Omron CX-Programmer project NewProject (CX-Programmer 9.61)

# PLC NewPLC1: CJ2M CPU31
I/O table (CPU CJ2M-CPU31): rack 0 slot 0 CJ1W-ID211; rack 0 slot 1 CJ1W-ID211; rack 0 slot 2 CJ1W-ID211; rack 0 slot 3 CJ1W-OD211; rack 0 slot 4 CJ1W-OD211; rack 0 slot 5 CJ1W-OD211; rack 0 slot 11 CJ2M-EIP21

## Global symbols (name address type ; comment)
0.00 BOOL  ; MASTER ON
0.01 BOOL  ; SW AUT/MAN
0.02 BOOL  ; PB START
0.03 BOOL  ; PB_EXECUTE
0.04 BOOL  ; PB RESET
0.06 BOOL  ; IN INV1 FAULT
0.07 BOOL  ; IN INV2 FAULT
0.08 BOOL  ; IN INV3 FAULT
0.09 BOOL  ; IN INV4 FAULT
0.10 BOOL  ; IN INV5 FAULT
0.11 BOOL  ; RUN INV1
0.12 BOOL  ; RUN INV2
0.13 BOOL  ; RUN INV3
0.14 BOOL  ; RUN INV4
0.15 BOOL  ; RUN INV5
10.00 BOOL  ; IR HMI PB FWD MOTOR 1
10.01 BOOL  ; IR HMI PB RVS MOTOR 1
10.02 BOOL  ; IR HMI PB FWD MOTOR2
10.03 BOOL  ; IR HMI PB RVS MOTOR2
10.04 BOOL  ; IR HMI PB STRAIGHT
10.05 BOOL  ; IR HMI PB TURN
10.06 BOOL  ; IR HMI PB FWD MOTOR4
10.07 BOOL  ; IR HMI PB RVS MOTOR4
10.08 BOOL  ; IR HMI PB FWD MOTOR5
10.09 BOOL  ; IR HMI PB RVS MOTOR 5
10.10 BOOL  ; IR HMI PB STP1 UP
10.11 BOOL  ; IR HMI PB STP1 DN
10.12 BOOL  ; IR HMI PB STP2 UP
10.13 BOOL  ; IR HMI PB STP2 DN
10.14 BOOL  ; IR HMI PB STP3 UP
10.15 BOOL  ; IR HMI PB STP3 DN
11.00 BOOL  ; AUTO READY
11.01 BOOL  ; MANUAL READY
11.04 BOOL  ; SET RFID ENABLED
11.05 BOOL  ; STRAIGHT CONV CONFIRM
11.06 BOOL  ; TURNING CONV CONFIRM
11.09 BOOL  ; 16.06
11.10 BOOL  ; DELETE ALL DATA
11.11 BOOL  ; ON/OFF YELLOW LAMP
11.13 BOOL  ; MATERIAL CANNOT ENTER SEGMEN 2
11.14 BOOL  ; DELETE 1 MEMORY ROTATE
11.15 BOOL  ; DELETE 1 MEMORY STRAIGHT
12.00 BOOL  ; MASTER OFF
13.02 BOOL  ; ROT_CONV_NEXT DATA
13.03 BOOL  ; ROT_CONV_PREV DATA
14.00 BOOL  ; IR MAN M1 FWD
14.01 BOOL  ; IR MAN M1 RVS
14.02 BOOL  ; IR MAN M2 FWD
14.03 BOOL  ; IR MAN M2 RVS
14.04 BOOL  ; IR MAN STRAIGHT ROT
14.05 BOOL  ; IR MAN TURN ROT
14.06 BOOL  ; IR MAN M4 FWD
14.07 BOOL  ; IR MAN M4 RVS
14.08 BOOL  ; IR MAN M5 FWD
14.09 BOOL  ; IR MAN M5 RVS
14.10 BOOL  ; IR MAN STP1 UP
14.11 BOOL  ; IR MAN STP1 DN
14.12 BOOL  ; IR MAN STP2 UP
14.13 BOOL  ; IR MAN STP2 DN
14.14 BOOL  ; IR MAN STP3 UP
14.15 BOOL  ; IR MAN STP3 DN
15.00 BOOL  ; IR RS UP STP1
15.01 BOOL  ; IR RS DN STP1
15.02 BOOL  ; IR RS UP STP2
15.03 BOOL  ; IR RS DN STP2
15.04 BOOL  ; IR RS UP STP3
15.05 BOOL  ; IR RS DN STP3
15.06 BOOL  ; IR FAULT CONFIRM
15.07 BOOL  ; IR OUT M1 FWD
15.08 BOOL  ; IR OUT M1 RVS
15.09 BOOL  ; IR OUT M2 FWD
15.10 BOOL  ; IR OUT M2 RVS
15.11 BOOL  ; IR OUT M3 FWD
15.12 BOOL  ; IR OUT M3 RVS
15.13 BOOL  ; IR OUT M4 FWD
15.14 BOOL  ; IR OUT M4 RVS
15.15 BOOL  ; IR OUT M5 FWD
16.00 BOOL  ; IR OUT M5 RVS
16.01 BOOL  ; IR PH1
16.02 BOOL  ; IR PH2
16.03 BOOL  ; IR PH3
16.04 BOOL  ; IR PH4
16.05 BOOL  ; IR PH5
16.06 BOOL  ; IR PH6
16.07 BOOL  ; IR PH7
16.08 BOOL  ; IR PH8
16.09 BOOL  ; IR PH9
16.10 BOOL  ; AUTO M1 FWD
16.11 BOOL  ; AUTO M2 FWD IN MATERIAL
16.12 BOOL  ; AUTO STP1 DOWN
16.13 BOOL  ; AUTO M2 FWD OUT MATERIAL
16.14 BOOL  ; AUTO STP1 UP
16.15 BOOL  ; AUTO STP2 DOWN
17.00 BOOL  ; AUTO ROLLER ROTARY FWD IN MATERIAL
17.01 BOOL  ; AUTO STP3 DOWN
17.02 BOOL  ; AUTO ROLLER ROTARY FWD OUT MATERIAL
17.03 BOOL  ; AUTO STP3 UP
17.04 BOOL  ; AUTO M4 FWD IN MATERIAL
17.06 BOOL  ; AUTO M5 FWD IN MATERIAL
17.07 BOOL  ; HOMEPOST
17.08 BOOL  ; IR MANUAL MODE
17.09 BOOL  ; AUTO STP2 UP
17.10 BOOL  ; MATERIAL STRAIGHT
17.11 BOOL  ; MATERIAL TURN
17.12 BOOL  ; IR RS UP STP ROTARY
17.13 BOOL  ; IR RS DN STP ROTARY
17.14 BOOL  ; IR LS TURN
17.15 BOOL  ; IR LS STRAIGHT
18.00 BOOL  ; IR HMI INDI M3 FWD
18.01 BOOL  ; IR HMI INDI M3 RVS
18.02 BOOL  ; IR HMI PB STP ROT UP
18.03 BOOL  ; IR HMI STP ROT DN
18.04 BOOL  ; IR MAN STP ROT UP
18.05 BOOL  ; IR MAN STP ROT DN
18.06 BOOL  ; AUTO DN STP ROTARY
18.07 BOOL  ; AUTO M3 TURN
18.08 BOOL  ; AUTO STP ROTARY UP
18.09 BOOL  ; CONFIRM BASE TURN
18.10 BOOL  ; AUTO STP2 DOWN TURN
18.11 BOOL  ; CONFIRM TRANFER MATERIAL
18.12 BOOL  ; AUTO STP ROT DN
18.13 BOOL  ; AUTO STP2 UP AFTER TRANSFER TURN
18.14 BOOL  ; AUTO M3 BACK STRAIGHT
18.15 BOOL  ; AUTO STP ROT UP AFTER TRANFER TURN
19.00 BOOL  ; MAN ROTARY TURN
19.01 BOOL  ; MAN ROTARY STRAIGHT
19.02 BOOL  ; STP ROT UP
19.03 BOOL  ; STP ROT UP
19.04 BOOL  ; IR MAN M ROLLER RVS
19.05 BOOL  ; IR MAN M ROLLER FWD
19.06 BOOL  ; IR HMI PB M ROLLER FWD
19.07 BOOL  ; IR HMI PB M ROLLER RVS
19.08 BOOL  ; SET LS STRAIGHT
19.09 BOOL  ; SET LS TURN
19.10 BOOL  ; SET STP ROT UP
19.11 BOOL  ; SET STP ROT UP
19.12 BOOL  ; SET STP ROT DN
19.13 BOOL  ; AUTO DELAY OFF M1
19.14 BOOL  ; SET HOMEPOST ALL
19.15 BOOL  ; AUTO ROLLER ROT RVS TRANFER MATERIAL
1.00 BOOL  ; PH1
1.01 BOOL  ; PH2
1.02 BOOL  ; PH3
1.03 BOOL  ; PH4
1.04 BOOL  ; EMERGENCY SHUTTER
1.05 BOOL  ; AIR PRESURE ON
1.06 BOOL  ; PH5
1.07 BOOL  ; RS UP STP2
1.08 BOOL  ; RS DN STP2
1.09 BOOL  ; PH6
1.10 BOOL  ; RS DN STP3
1.11 BOOL  ; RS UP STP3
1.12 BOOL  ; RS UP STP ROTARY
1.13 BOOL  ; RS DN STP ROTARY
1.14 BOOL  ; LS TURN
1.15 BOOL  ; LS STRAIGHT
20.00 BOOL  ; SAVE 1
20.01 BOOL  ; SAVE 2
20.02 BOOL  ; HMI IN NO BLOWING
20.03 BOOL  ; CONFIRM NO BLOWING
20.04 BOOL  ; AIR SOURCE OFF CONFIRM
20.05 BOOL  ; SET DELAY STP3 UP
20.06 BOOL  ; DON'T CONFIRM
20.07 BOOL  ; ROT RUN TURN
20.08 BOOL  ; SET OF M5
20.09 BOOL  ; SET OFF M1
20.10 BOOL  ; LONG MATERIAL WAITING IN ROTARY
20.11 BOOL  ; DELAY OFF RVS ROLLER
20.12 BOOL  ; IR LAST DATA
20.13 BOOL  ; MATERIAL WAIT ON CONV 1
20.14 BOOL  ; STP2 UP WAIT LONG MATERIAL
20.15 BOOL  ; STP2 CAN'T UP
2.00 BOOL  ; PH7
2.01 BOOL  ; PH8
2.02 BOOL  ; PH9
2.03 BOOL  ; PH9
2.04 BOOL  ; INTERLOCK BLOWING DOOR NOT OPEN
2.05 BOOL  ; INTERLOCK BLOWING PHOTOSENSOR
2.12 BOOL  ; RS DN STP1
2.13 BOOL  ; RS UP STP1
3.00 BOOL  ; SOL UP STP1
3.01 BOOL  ; SOL DN STP1
3.02 BOOL  ; SOL UP STP2
3.03 BOOL  ; SOL DN STP2
3.04 BOOL  ; SOL UP STP3
3.05 BOOL  ; SOL DN STP3
3.08 BOOL  ; TOWER LAMP GREEN
3.09 BOOL  ; TOWER LAMP YELLOW
3.10 BOOL  ; TOWER LAMP RED
3.11 BOOL  ; OUT RESET INV1
3.12 BOOL  ; OUT RESET INV2
3.13 BOOL  ; OUT RESET INV3
3.14 BOOL  ; OUT RESET INV4
3.15 BOOL  ; OUT RESET INV5
4.00 BOOL  ; BUZZER
4.01 BOOL  ; AUTORUN LAMP
4.02 BOOL  ; INDILAMP YELLOW
4.03 BOOL  ; FAULT LAMP
4.04 BOOL  ; OUT M1 FWD
4.05 BOOL  ; OUT M1 RVS
4.06 BOOL  ; OUT M2 FWD
4.07 BOOL  ; OUT M2 RVS
4.08 BOOL  ; OUT M3 TURN
4.09 BOOL  ; OUT M3 STRAIGHT
4.10 BOOL  ; OUT M4 FWD
4.11 BOOL  ; OUT M4 RVS
4.12 BOOL  ; OUT M5 FWD
4.13 BOOL  ; OUT M5 RVS
4.14 BOOL  ; KONTAKTOR M4
4.15 BOOL  ; KONTAKTOR M5
5.00 BOOL  ; SOL UP STP ROT
5.01 BOOL  ; SOL DN STP ROT
5.02 BOOL  ; OUT RELAY BRAKE
5.03 BOOL  ; OUT M ROLLER FWD
5.04 BOOL  ; OUT M ROLLER RVS
5.05 BOOL  ; BLOWING NO ROTATE
5.15 BOOL  ; chiyoda
99.00 BOOL  ; MASTER ON
99.01 BOOL  ; MASTER OFF
99.02 BOOL  ; IR_FAULT_CONFIRM
D1000 CHANNEL  ; READ DATA FROM RFID
D1002 CHANNEL  ; INPUT DATA WORD 1
D1003 CHANNEL  ; INPUT DATA WORD 2
D1010 CHANNEL  ; ID RECODED 1
D1011 CHANNEL  ; ID RECORDED2
D1093 CHANNEL  ; STACK LOCATION
D1450 CHANNEL  ; DATA INDIRECT
D1460 CHANNEL  ; DATA INDIRECT
D1800 CHANNEL  ; DATA INPUT
D1820 CHANNEL  ; DATA INPUT
D2000 CHANNEL  ; MEMORY 1 NO BLOWING
D2002 CHANNEL  ; MEEMORY 2 NO BLOWING
D2004 CHANNEL  ; MEMORY NO 3 NO BLOWING
D2006 CHANNEL  ; MEMORY 4 NO BLOWING
D2008 CHANNEL  ; MEMORY 5 NO BLOWING
D2010 CHANNEL  ; MEMORY 6 NO BLOWING
D2012 CHANNEL  ; MEMORY 7 NO BLOWING
D2014 CHANNEL  ; MEMORY 8 NO BLOWING
D2016 CHANNEL  ; MEMORY 9 NO BLOWING
D2018 CHANNEL  ; MEMORY 10 NO BLOWING
D3000 CHANNEL  ; LAST DATA ACTION
D50 CHANNEL  ; ID RECORDED1
D51 CHANNEL  ; ID RECORDED2
D90 CHANNEL  ; DATA STRAIGHT STACK
D91 CHANNEL  ; DATA 2X STRAIGHT STACK
T0001 BOOL  ; DELAY ON M1
T0002 BOOL  ; DELAY OFF M1
T0003 BOOL  ; DELAY OFF M2 OUT MATERIAL
T0004 BOOL  ; DELAY DOWN STP3
T0005 BOOL  ; DELAY OFF MOTOR ROLLER
T0006 BOOL  ; DELAY UP STP 3
T0007 BOOL  ; DELAY STP1 DOWN
T0008 BOOL  ; DELAY TURN
T0009 BOOL  ; DELAY STP3 UP
T0010 BOOL  ; DELAY SAFETY OFF BY SELF
T0011 BOOL  ; DELAY SAFETY OFF BY SELF M2
T0012 BOOL  ; DELAY SAFETY OFF BY SELF
T0013 BOOL  ; DELAY OFF BUTTON NO ROTATE BLOWING
T0014 BOOL  ; DELAY OFF SET ROTARY MANUAL
T0015 BOOL  ; DELAY OFF M5
T0016 BOOL  ; DELAY OFF M1
T0017 BOOL  ; DELAY OFF SET HOMEPOST
T0019 BOOL  ; DELAY OFF ROLLER RVS
W0.00 BOOL  ; HMI_OUT_MASTER ON
W0.01 BOOL  ; HMI_HOMEPOST
W0.02 BOOL  ; HMI_OUT_AUTORUN
W0.03 BOOL  ; HMI_OUT_FAULT
W0.04 BOOL  ; HMI_OUT_READER ON
W0.05 BOOL  ; HMI_PB_M1_FWD
W0.06 BOOL  ; HMI_PB_M1_RVS
W0.07 BOOL  ; HMI_PB_M2_FWD
W0.08 BOOL  ; HMI_PB_M2_RVS
W0.09 BOOL  ; HMI_PB_M3_FWD
W0.10 BOOL  ; HMI_PB_M3_RVS
W0.11 BOOL  ; HMI_PB_M4_FWD
W0.12 BOOL  ; HMI_PB_M4_RVS
W0.13 BOOL  ; HMI_PB_M5_FWD
W0.14 BOOL  ; HMI_PB_M5_RVS
W0.15 BOOL  ; HMI_PB_STP1_UP
W10.00 BOOL  ; HMI_IN_READ ENABLE
W11.06 BOOL  ; TURN BLOWING
W1.00 BOOL  ; HMI_PB_STP1_DN
W1.01 BOOL  ; HMI_PB_STP2_UP
W1.02 BOOL  ; HMI_PB_STP2_DN
W1.03 BOOL  ; HMI_PB_STP3_UP
W1.04 BOOL  ; HMI_PB_STP3_DN
W1.05 BOOL  ; OUT HMI INDI M1 FWD
W1.06 BOOL  ; OUT HMI INDI M1 RVS
W1.07 BOOL  ; OUT HMI INDI M2 FWD
W1.08 BOOL  ; OUT HMI INDI M2 RVS
W1.09 BOOL  ; OUT HMI INDI M3 FWD
W1.10 BOOL  ; OUT HMI INDI M3 RVS
W1.11 BOOL  ; OUT HMI INDI M4 FWD
W1.12 BOOL  ; OUT HMI INDI M4 RVS
W1.13 BOOL  ; OUT HMI INDI M5 FWD
W1.14 BOOL  ; OUT HMI INDI M5 RVS
W1.15 BOOL  ; OUT HMI INDI STP1 UP
W2.00 BOOL  ; OUT HMI INDI STP1 DN
W2.01 BOOL  ; OUT HMI INDI STP2 UP
W2.02 BOOL  ; OUT HMI INDI STP2 DN
W2.03 BOOL  ; OUT HMI INDI STP3 UP
W2.04 BOOL  ; OUT HMI INDI STP3 DN
W2.05 BOOL  ; OUT HMI INDI MASTER ON
W2.06 BOOL  ; OUT HMI INDI MANUAL
W2.07 BOOL  ; HMI FAULT INV1
W2.08 BOOL  ; HMI FAULT INV2
W2.09 BOOL  ; HMI FAULT INV3
W2.10 BOOL  ; HMI FAULT INV4
W2.11 BOOL  ; HMI FAULT INV5
W2.12 BOOL  ; HMI MASTER OFF
W2.13 BOOL  ; HMI RESET FAULT
W2.14 BOOL  ; HMI NOTIF EMERGENCY
W2.15 BOOL  ; HMI INDI CONV STRAIGHT
W3.00 BOOL  ; HMI INDI CONV ROTATE
W3.01 BOOL  ; HMI PB STP ROT UP
W3.02 BOOL  ; HMI PB STP ROT DN
W3.03 BOOL  ; OUT HMI INDI STP ROT UP
W3.04 BOOL  ; OUT HMI INDI STP ROT DN
W3.05 BOOL  ; HMI PB M ROLLER FWD
W3.06 BOOL  ; HMI PB M ROLLER RVS
W3.07 BOOL  ; AIR OFF NOTIF
W3.08 BOOL  ; HMI INDI M ROLLER FWD
W3.09 BOOL  ; HMI INDI M ROLLER RVS
W3.10 BOOL  ; HMI MATERIAL ROTATE AND NO ROTATE
W3.11 BOOL  ; HMI PB HOMEPOST
FILTERING_DATA1 FOR
FORJUGA FOR
Incoming_Data DATAMOVEMENT
LURUS_GAES DATAMOVEMENT
NO_BLOWING_SEQUENCE NO_BLOWING

## Program NewProgram1 (cyclic task 0)
Local symbols
P_0n BOOL

### Section MAIN

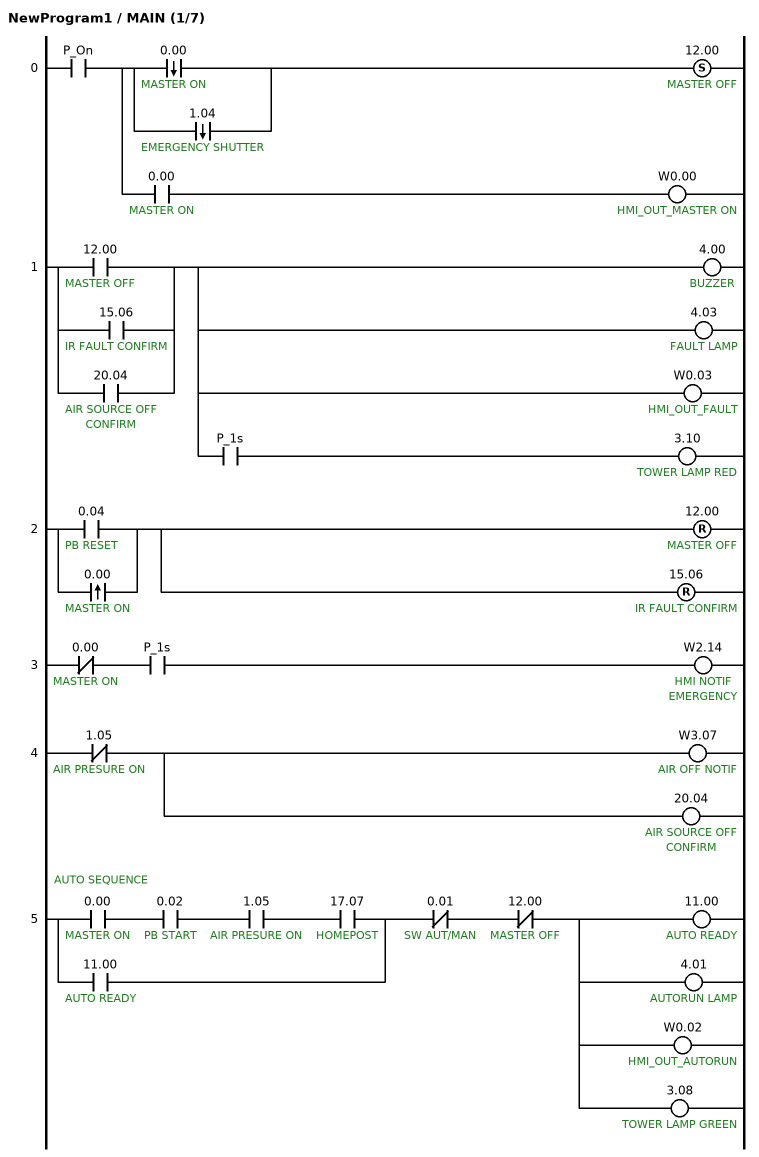
; rung 0
LD P_On
OUT TR0
%LD 0.00  ; MASTER ON
%OR 1.04  ; EMERGENCY SHUTTER
ANDLD
SET 12.00  ; MASTER OFF
LD TR0
AND 0.00  ; MASTER ON
OUT W0.00  ; HMI_OUT_MASTER ON
; rung 1
LD 12.00  ; MASTER OFF
OR 15.06  ; IR FAULT CONFIRM
OR 20.04  ; AIR SOURCE OFF CONFIRM
OUT 4.00  ; BUZZER
OUT 4.03  ; FAULT LAMP
OUT W0.03  ; HMI_OUT_FAULT
AND P_1s
OUT 3.10  ; TOWER LAMP RED
; rung 2
LD 0.04  ; PB RESET
@OR 0.00  ; MASTER ON
RSET 12.00  ; MASTER OFF
RSET 15.06  ; IR FAULT CONFIRM
; rung 3
LDNOT 0.00  ; MASTER ON
AND P_1s
OUT W2.14  ; HMI NOTIF EMERGENCY
; rung 4
LDNOT 1.05  ; AIR PRESURE ON
OUT W3.07  ; AIR OFF NOTIF
OUT 20.04  ; AIR SOURCE OFF CONFIRM
; rung 5: AUTO SEQUENCE
LD 0.00  ; MASTER ON
AND 0.02  ; PB START
AND 1.05  ; AIR PRESURE ON
AND 17.07  ; HOMEPOST
OR 11.00  ; AUTO READY
ANDNOT 0.01  ; SW AUT/MAN
ANDNOT 12.00  ; MASTER OFF
OUT 11.00  ; AUTO READY
OUT 4.01  ; AUTORUN LAMP
OUT W0.02  ; HMI_OUT_AUTORUN
OUT 3.08  ; TOWER LAMP GREEN

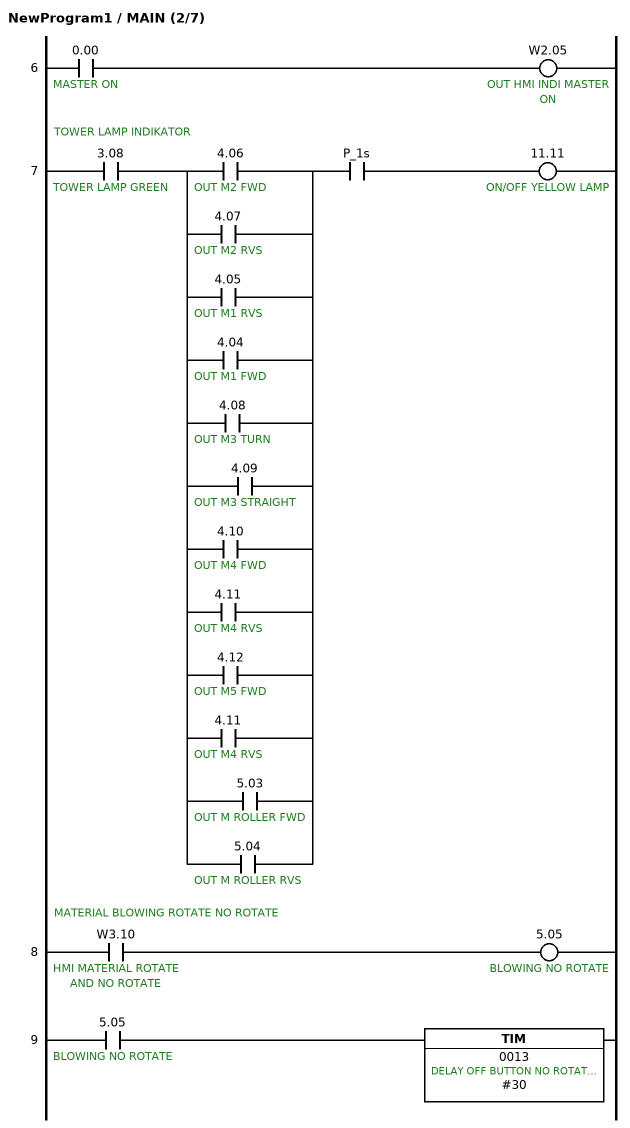
; rung 6
LD 0.00  ; MASTER ON
OUT W2.05  ; OUT HMI INDI MASTER ON
; rung 7: TOWER LAMP INDIKATOR
LD 3.08  ; TOWER LAMP GREEN
LD 4.06  ; OUT M2 FWD
OR 4.07  ; OUT M2 RVS
OR 4.05  ; OUT M1 RVS
OR 4.04  ; OUT M1 FWD
OR 4.08  ; OUT M3 TURN
OR 4.09  ; OUT M3 STRAIGHT
OR 4.10  ; OUT M4 FWD
OR 4.11  ; OUT M4 RVS
OR 4.12  ; OUT M5 FWD
OR 4.11  ; OUT M4 RVS
OR 5.03  ; OUT M ROLLER FWD
OR 5.04  ; OUT M ROLLER RVS
ANDLD
AND P_1s
OUT 11.11  ; ON/OFF YELLOW LAMP
; rung 8: MATERIAL BLOWING ROTATE NO ROTATE
LD W3.10  ; HMI MATERIAL ROTATE AND NO ROTATE
OUT 5.05  ; BLOWING NO ROTATE
; rung 9
LD 5.05  ; BLOWING NO ROTATE
TIM 0013 #30  ; DELAY OFF BUTTON NO ROTATE BLOWING

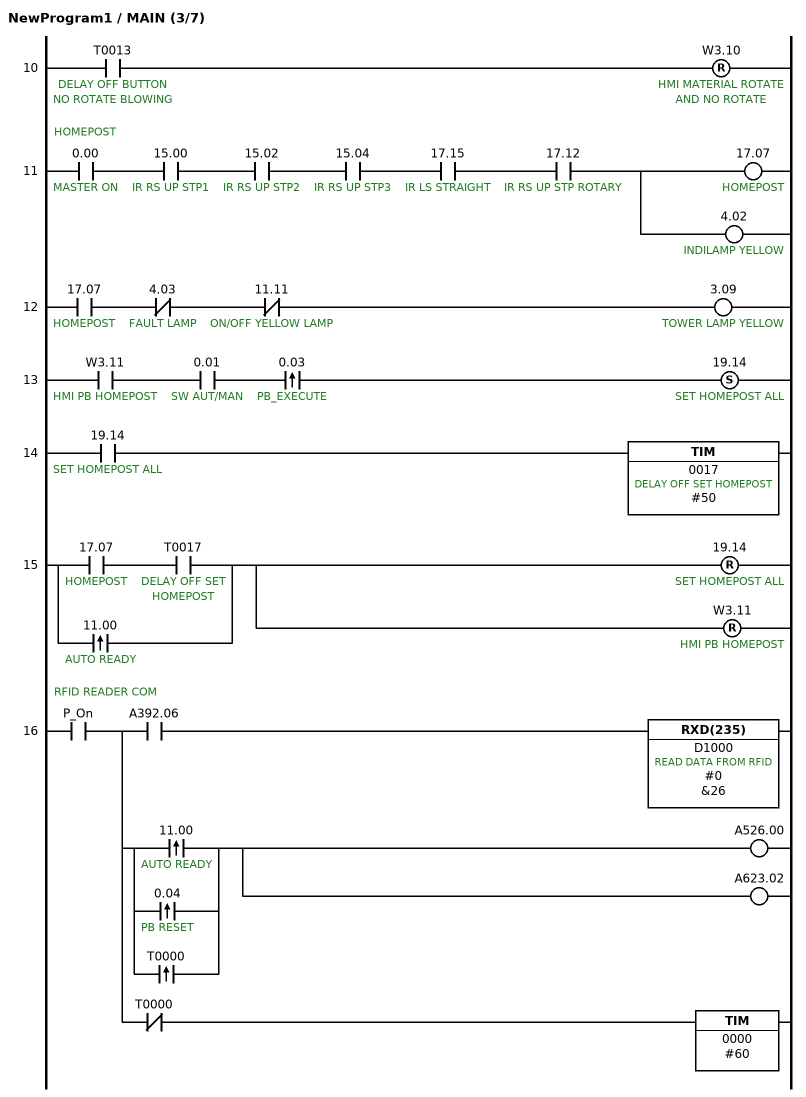
; rung 10
LD T0013  ; DELAY OFF BUTTON NO ROTATE BLOWING
RSET W3.10  ; HMI MATERIAL ROTATE AND NO ROTATE
; rung 11: HOMEPOST
LD 0.00  ; MASTER ON
AND 15.00  ; IR RS UP STP1
AND 15.02  ; IR RS UP STP2
AND 15.04  ; IR RS UP STP3
AND 17.15  ; IR LS STRAIGHT
AND 17.12  ; IR RS UP STP ROTARY
OUT 17.07  ; HOMEPOST
OUT 4.02  ; INDILAMP YELLOW
; rung 12
LD 17.07  ; HOMEPOST
ANDNOT 4.03  ; FAULT LAMP
ANDNOT 11.11  ; ON/OFF YELLOW LAMP
OUT 3.09  ; TOWER LAMP YELLOW
; rung 13
LD W3.11  ; HMI PB HOMEPOST
AND 0.01  ; SW AUT/MAN
@AND 0.03  ; PB_EXECUTE
SET 19.14  ; SET HOMEPOST ALL
; rung 14
LD 19.14  ; SET HOMEPOST ALL
TIM 0017 #50  ; DELAY OFF SET HOMEPOST
; rung 15
LD 17.07  ; HOMEPOST
AND T0017  ; DELAY OFF SET HOMEPOST
@OR 11.00  ; AUTO READY
RSET 19.14  ; SET HOMEPOST ALL
RSET W3.11  ; HMI PB HOMEPOST
; rung 16: RFID READER COM
LD P_On
OUT TR0
AND A392.06
RXD(235) D1000 #0 &26  ; READ DATA FROM RFID
LD TR0
@LD 11.00  ; AUTO READY
@OR 0.04  ; PB RESET
@OR T0000
ANDLD
OUT A526.00
OUT A623.02
LD TR0
ANDNOT T0000
TIM 0000 #60

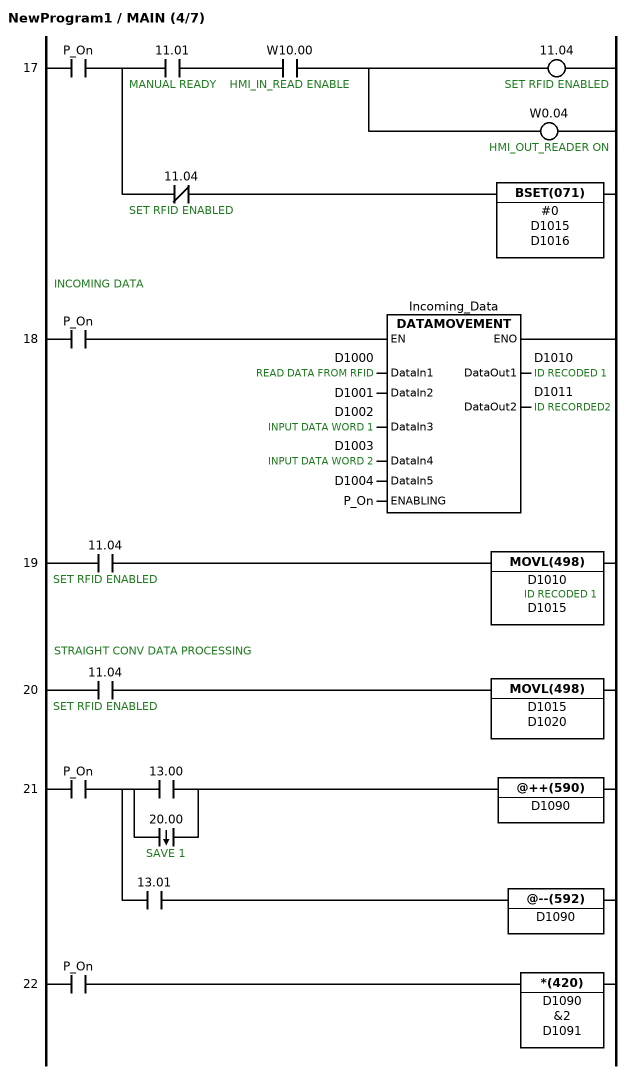
; rung 17
LD P_On
OUT TR0
AND 11.01  ; MANUAL READY
AND W10.00  ; HMI_IN_READ ENABLE
OUT 11.04  ; SET RFID ENABLED
OUT W0.04  ; HMI_OUT_READER ON
LD TR0
ANDNOT 11.04  ; SET RFID ENABLED
BSET(071) #0 D1015 D1016
; rung 18: INCOMING DATA
LD P_On
CALL Incoming_Data : DATAMOVEMENT (DataIn1 := D1000, DataIn2 := D1001, DataIn3 := D1002, DataIn4 := D1003, DataIn5 := D1004, ENABLING := P_On, DataOut1 => D1010, DataOut2 => D1011)  ; READ DATA FROM RFID, INPUT DATA WORD 1, INPUT DATA WORD 2, ID RECODED 1, ID RECORDED2
; rung 19
LD 11.04  ; SET RFID ENABLED
MOVL(498) D1010 D1015  ; ID RECODED 1
; rung 20: STRAIGHT CONV DATA PROCESSING
LD 11.04  ; SET RFID ENABLED
MOVL(498) D1015 D1020
; rung 21
LD P_On
OUT TR0
LD 13.00
%OR 20.00  ; SAVE 1
ANDLD
@++(590) D1090
LD TR0
AND 13.01
@--(592) D1090
; rung 22
LD P_On
*(420) D1090 &2 D1091

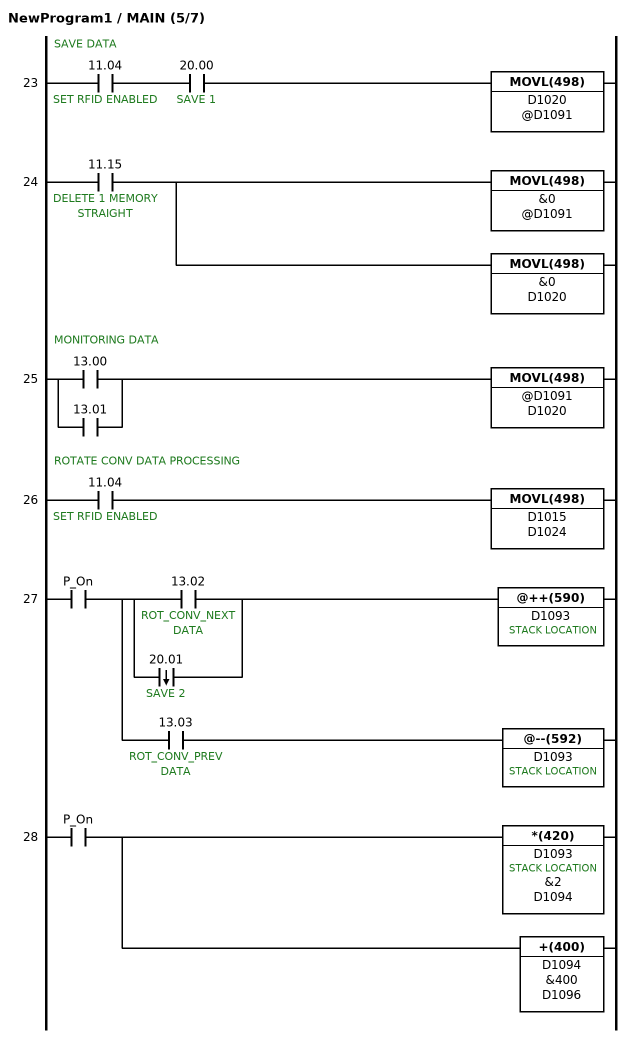
; rung 23: SAVE DATA
LD 11.04  ; SET RFID ENABLED
AND 20.00  ; SAVE 1
MOVL(498) D1020 @D1091
; rung 24
LD 11.15  ; DELETE 1 MEMORY STRAIGHT
MOVL(498) &0 @D1091
MOVL(498) &0 D1020
; rung 25: MONITORING DATA
LD 13.00
OR 13.01
MOVL(498) @D1091 D1020
; rung 26: ROTATE CONV DATA PROCESSING
LD 11.04  ; SET RFID ENABLED
MOVL(498) D1015 D1024
; rung 27
LD P_On
OUT TR0
LD 13.02  ; ROT_CONV_NEXT DATA
%OR 20.01  ; SAVE 2
ANDLD
@++(590) D1093  ; STACK LOCATION
LD TR0
AND 13.03  ; ROT_CONV_PREV DATA
@--(592) D1093  ; STACK LOCATION
; rung 28
LD P_On
*(420) D1093 &2 D1094  ; STACK LOCATION
+(400) D1094 &400 D1096

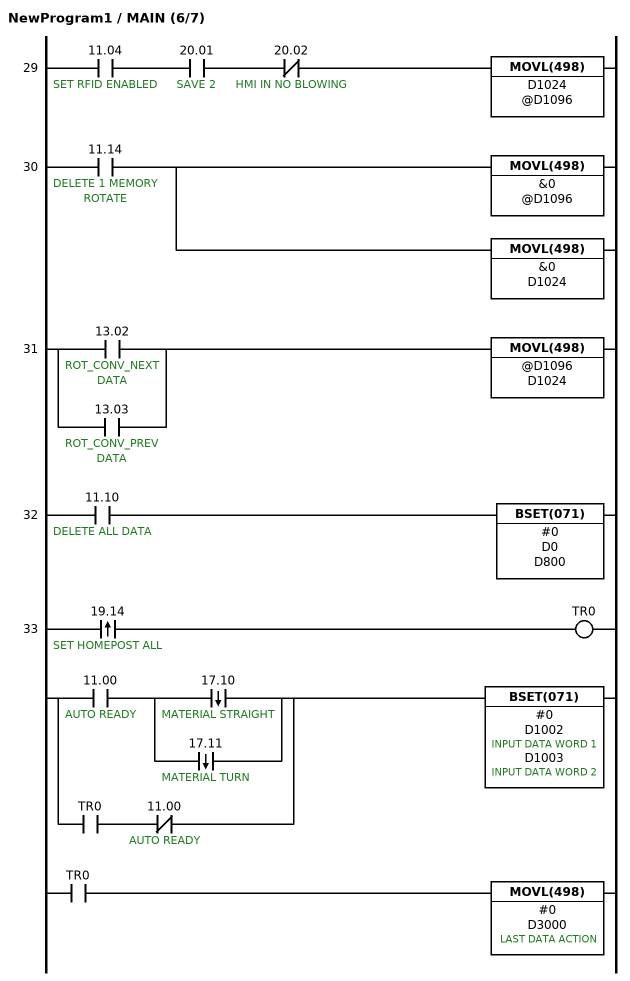
; rung 29
LD 11.04  ; SET RFID ENABLED
AND 20.01  ; SAVE 2
ANDNOT 20.02  ; HMI IN NO BLOWING
MOVL(498) D1024 @D1096
; rung 30
LD 11.14  ; DELETE 1 MEMORY ROTATE
MOVL(498) &0 @D1096
MOVL(498) &0 D1024
; rung 31
LD 13.02  ; ROT_CONV_NEXT DATA
OR 13.03  ; ROT_CONV_PREV DATA
MOVL(498) @D1096 D1024
; rung 32
LD 11.10  ; DELETE ALL DATA
BSET(071) #0 D0 D800
; rung 33
LD 11.00  ; AUTO READY
%LD 17.10  ; MATERIAL STRAIGHT
%OR 17.11  ; MATERIAL TURN
ANDLD
@LD 19.14  ; SET HOMEPOST ALL
OUT TR0
ANDNOT 11.00  ; AUTO READY
ORLD
BSET(071) #0 D1002 D1003  ; INPUT DATA WORD 1, INPUT DATA WORD 2
LD TR0
MOVL(498) #0 D3000  ; LAST DATA ACTION

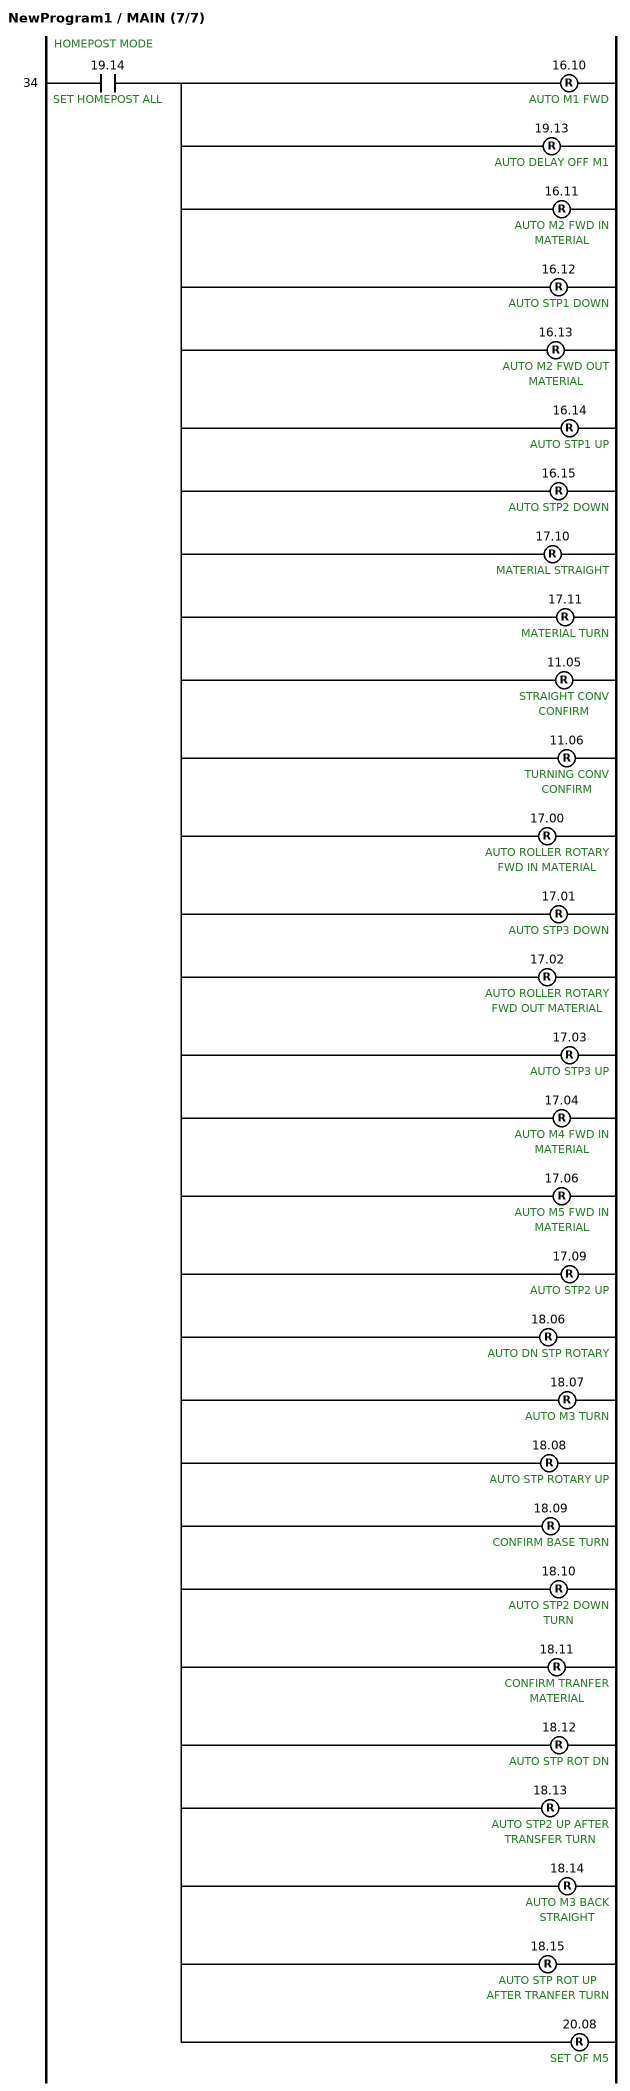
; rung 34: HOMEPOST MODE
LD 19.14  ; SET HOMEPOST ALL
RSET 16.10  ; AUTO M1 FWD
RSET 19.13  ; AUTO DELAY OFF M1
RSET 16.11  ; AUTO M2 FWD IN MATERIAL
RSET 16.12  ; AUTO STP1 DOWN
RSET 16.13  ; AUTO M2 FWD OUT MATERIAL
RSET 16.14  ; AUTO STP1 UP
RSET 16.15  ; AUTO STP2 DOWN
RSET 17.10  ; MATERIAL STRAIGHT
RSET 17.11  ; MATERIAL TURN
RSET 11.05  ; STRAIGHT CONV CONFIRM
RSET 11.06  ; TURNING CONV CONFIRM
RSET 17.00  ; AUTO ROLLER ROTARY FWD IN MATERIAL
RSET 17.01  ; AUTO STP3 DOWN
RSET 17.02  ; AUTO ROLLER ROTARY FWD OUT MATERIAL
RSET 17.03  ; AUTO STP3 UP
RSET 17.04  ; AUTO M4 FWD IN MATERIAL
RSET 17.06  ; AUTO M5 FWD IN MATERIAL
RSET 17.09  ; AUTO STP2 UP
RSET 18.06  ; AUTO DN STP ROTARY
RSET 18.07  ; AUTO M3 TURN
RSET 18.08  ; AUTO STP ROTARY UP
RSET 18.09  ; CONFIRM BASE TURN
RSET 18.10  ; AUTO STP2 DOWN TURN
RSET 18.11  ; CONFIRM TRANFER MATERIAL
RSET 18.12  ; AUTO STP ROT DN
RSET 18.13  ; AUTO STP2 UP AFTER TRANSFER TURN
RSET 18.14  ; AUTO M3 BACK STRAIGHT
RSET 18.15  ; AUTO STP ROT UP AFTER TRANFER TURN
RSET 20.08  ; SET OF M5

### Section CONV

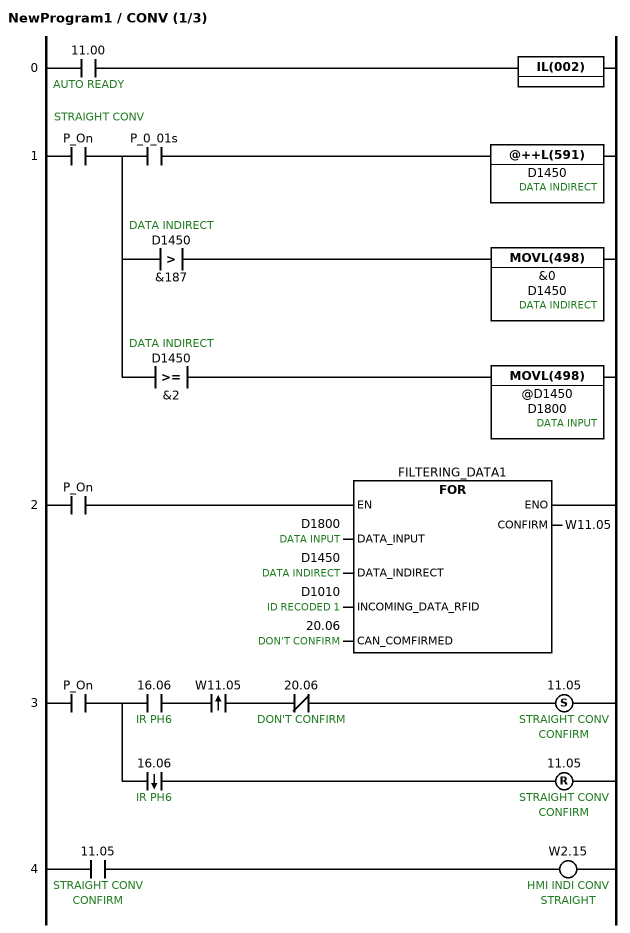
; rung 0
LD 11.00  ; AUTO READY
IL(002)
; rung 1: STRAIGHT CONV
LD P_On
OUT TR0
AND P_0_01s
@++L(591) D1450  ; DATA INDIRECT
LD TR0
AND>(320) D1450 &187  ; DATA INDIRECT
MOVL(498) &0 D1450  ; DATA INDIRECT
LD TR0
AND>=(325) D1450 &2  ; DATA INDIRECT
MOVL(498) @D1450 D1800  ; DATA INPUT
; rung 2
LD P_On
CALL FILTERING_DATA1 : FOR (DATA_INPUT := D1800, DATA_INDIRECT := D1450, INCOMING_DATA_RFID := D1010, CAN_COMFIRMED := 20.06, CONFIRM => W11.05)  ; DATA INPUT, DATA INDIRECT, ID RECODED 1, DON'T CONFIRM
; rung 3
LD P_On
OUT TR0
AND 16.06  ; IR PH6
@AND W11.05
ANDNOT 20.06  ; DON'T CONFIRM
SET 11.05  ; STRAIGHT CONV CONFIRM
LD TR0
%AND 16.06  ; IR PH6
RSET 11.05  ; STRAIGHT CONV CONFIRM
; rung 4
LD 11.05  ; STRAIGHT CONV CONFIRM
OUT W2.15  ; HMI INDI CONV STRAIGHT

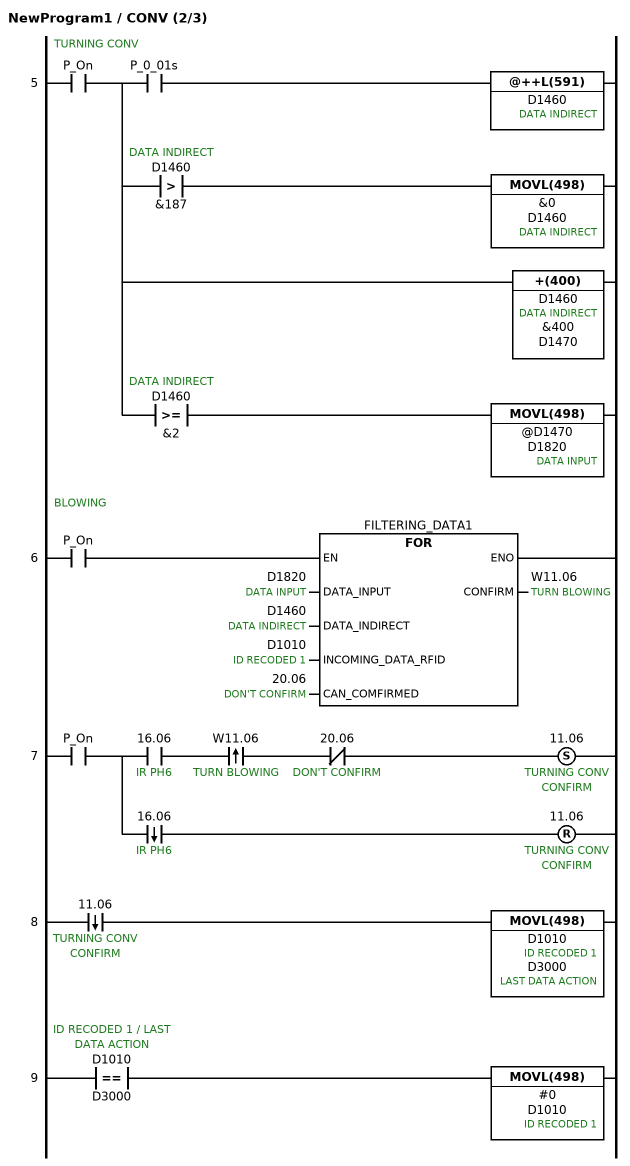
; rung 5: TURNING CONV
LD P_On
OUT TR0
AND P_0_01s
@++L(591) D1460  ; DATA INDIRECT
LD TR0
AND>(320) D1460 &187  ; DATA INDIRECT
MOVL(498) &0 D1460  ; DATA INDIRECT
LD TR0
+(400) D1460 &400 D1470  ; DATA INDIRECT
AND>=(325) D1460 &2  ; DATA INDIRECT
MOVL(498) @D1470 D1820  ; DATA INPUT
; rung 6: BLOWING
LD P_On
CALL FILTERING_DATA1 : FOR (DATA_INPUT := D1820, DATA_INDIRECT := D1460, INCOMING_DATA_RFID := D1010, CAN_COMFIRMED := 20.06, CONFIRM => W11.06)  ; DATA INPUT, DATA INDIRECT, ID RECODED 1, DON'T CONFIRM, TURN BLOWING
; rung 7
LD P_On
OUT TR0
AND 16.06  ; IR PH6
@AND W11.06  ; TURN BLOWING
ANDNOT 20.06  ; DON'T CONFIRM
SET 11.06  ; TURNING CONV CONFIRM
LD TR0
%AND 16.06  ; IR PH6
RSET 11.06  ; TURNING CONV CONFIRM
; rung 8
%LD 11.06  ; TURNING CONV CONFIRM
MOVL(498) D1010 D3000  ; ID RECODED 1, LAST DATA ACTION
; rung 9
LD=L(301) D1010 D3000  ; ID RECODED 1, LAST DATA ACTION
MOVL(498) #0 D1010  ; ID RECODED 1

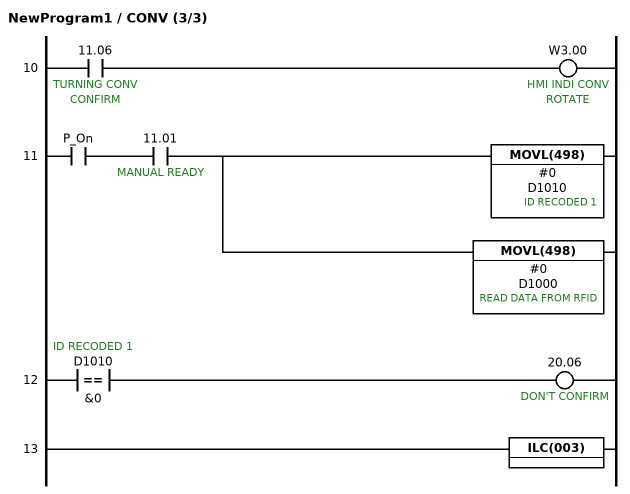
; rung 10
LD 11.06  ; TURNING CONV CONFIRM
OUT W3.00  ; HMI INDI CONV ROTATE
; rung 11
LD P_On
AND 11.01  ; MANUAL READY
MOVL(498) #0 D1010  ; ID RECODED 1
MOVL(498) #0 D1000  ; READ DATA FROM RFID
; rung 12
LD=(300) D1010 &0  ; ID RECODED 1
OUT 20.06  ; DON'T CONFIRM
; rung 13
ILC(003)

### Section MANUAL_SEQ

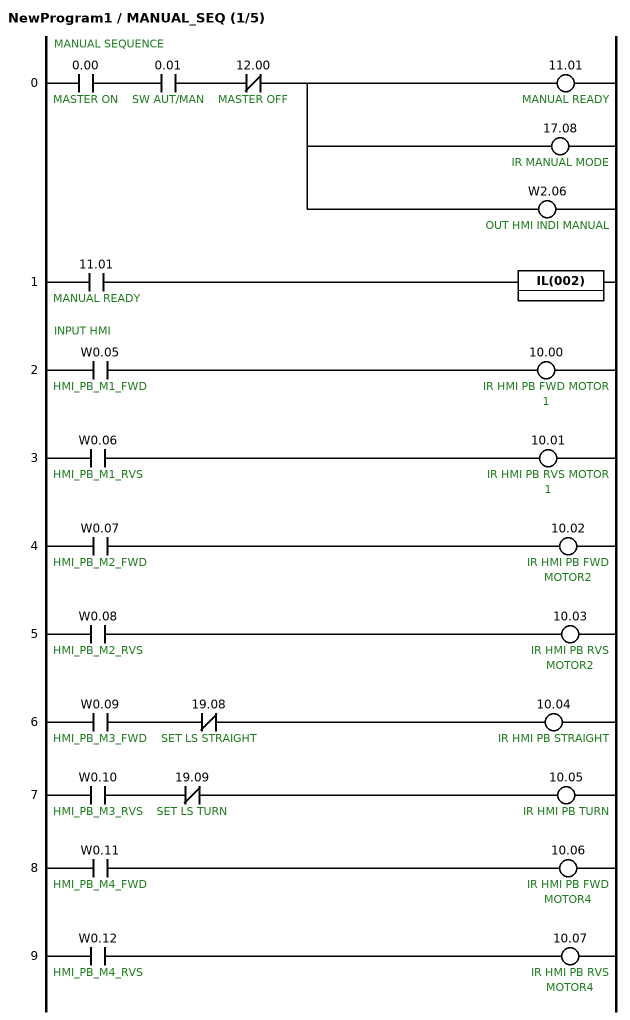
; rung 0: MANUAL SEQUENCE
LD 0.00  ; MASTER ON
AND 0.01  ; SW AUT/MAN
ANDNOT 12.00  ; MASTER OFF
OUT 11.01  ; MANUAL READY
OUT 17.08  ; IR MANUAL MODE
OUT W2.06  ; OUT HMI INDI MANUAL
; rung 1
LD 11.01  ; MANUAL READY
IL(002)
; rung 2: INPUT HMI
LD W0.05  ; HMI_PB_M1_FWD
OUT 10.00  ; IR HMI PB FWD MOTOR 1
; rung 3
LD W0.06  ; HMI_PB_M1_RVS
OUT 10.01  ; IR HMI PB RVS MOTOR 1
; rung 4
LD W0.07  ; HMI_PB_M2_FWD
OUT 10.02  ; IR HMI PB FWD MOTOR2
; rung 5
LD W0.08  ; HMI_PB_M2_RVS
OUT 10.03  ; IR HMI PB RVS MOTOR2
; rung 6
LD W0.09  ; HMI_PB_M3_FWD
ANDNOT 19.08  ; SET LS STRAIGHT
OUT 10.04  ; IR HMI PB STRAIGHT
; rung 7
LD W0.10  ; HMI_PB_M3_RVS
ANDNOT 19.09  ; SET LS TURN
OUT 10.05  ; IR HMI PB TURN
; rung 8
LD W0.11  ; HMI_PB_M4_FWD
OUT 10.06  ; IR HMI PB FWD MOTOR4
; rung 9
LD W0.12  ; HMI_PB_M4_RVS
OUT 10.07  ; IR HMI PB RVS MOTOR4

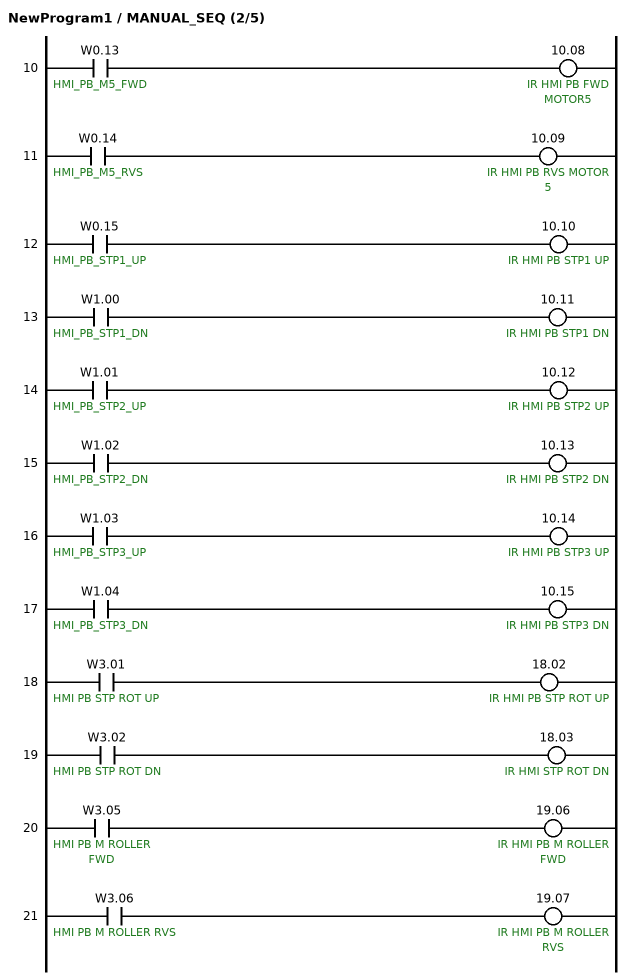
; rung 10
LD W0.13  ; HMI_PB_M5_FWD
OUT 10.08  ; IR HMI PB FWD MOTOR5
; rung 11
LD W0.14  ; HMI_PB_M5_RVS
OUT 10.09  ; IR HMI PB RVS MOTOR 5
; rung 12
LD W0.15  ; HMI_PB_STP1_UP
OUT 10.10  ; IR HMI PB STP1 UP
; rung 13
LD W1.00  ; HMI_PB_STP1_DN
OUT 10.11  ; IR HMI PB STP1 DN
; rung 14
LD W1.01  ; HMI_PB_STP2_UP
OUT 10.12  ; IR HMI PB STP2 UP
; rung 15
LD W1.02  ; HMI_PB_STP2_DN
OUT 10.13  ; IR HMI PB STP2 DN
; rung 16
LD W1.03  ; HMI_PB_STP3_UP
OUT 10.14  ; IR HMI PB STP3 UP
; rung 17
LD W1.04  ; HMI_PB_STP3_DN
OUT 10.15  ; IR HMI PB STP3 DN
; rung 18
LD W3.01  ; HMI PB STP ROT UP
OUT 18.02  ; IR HMI PB STP ROT UP
; rung 19
LD W3.02  ; HMI PB STP ROT DN
OUT 18.03  ; IR HMI STP ROT DN
; rung 20
LD W3.05  ; HMI PB M ROLLER FWD
OUT 19.06  ; IR HMI PB M ROLLER FWD
; rung 21
LD W3.06  ; HMI PB M ROLLER RVS
OUT 19.07  ; IR HMI PB M ROLLER RVS

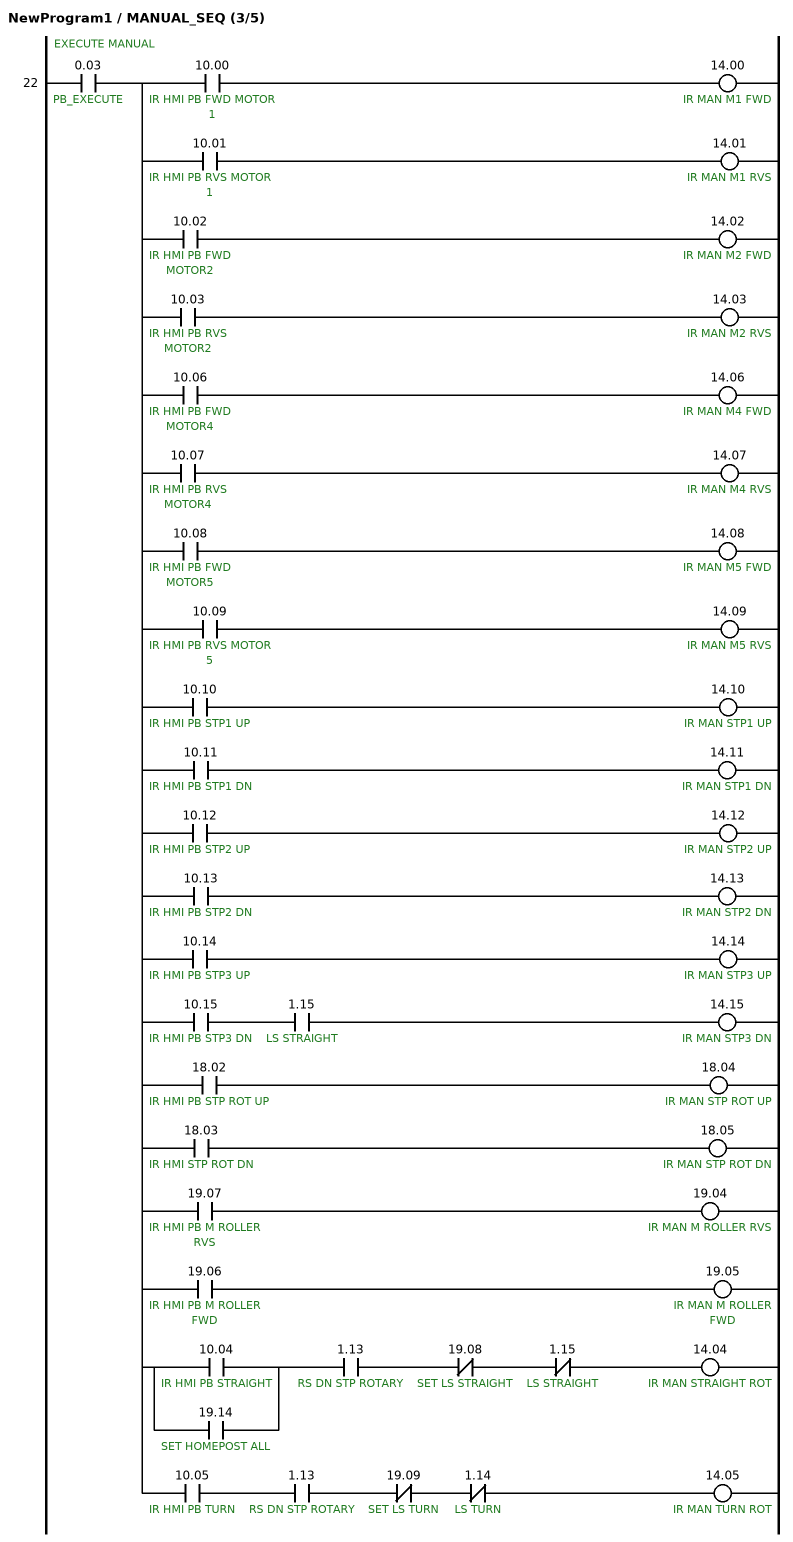
; rung 22: EXECUTE MANUAL
LD 0.03  ; PB_EXECUTE
OUT TR0
AND 10.00  ; IR HMI PB FWD MOTOR 1
OUT 14.00  ; IR MAN M1 FWD
LD TR0
AND 10.01  ; IR HMI PB RVS MOTOR 1
OUT 14.01  ; IR MAN M1 RVS
LD TR0
AND 10.02  ; IR HMI PB FWD MOTOR2
OUT 14.02  ; IR MAN M2 FWD
LD TR0
AND 10.03  ; IR HMI PB RVS MOTOR2
OUT 14.03  ; IR MAN M2 RVS
LD TR0
AND 10.06  ; IR HMI PB FWD MOTOR4
OUT 14.06  ; IR MAN M4 FWD
LD TR0
AND 10.07  ; IR HMI PB RVS MOTOR4
OUT 14.07  ; IR MAN M4 RVS
LD TR0
AND 10.08  ; IR HMI PB FWD MOTOR5
OUT 14.08  ; IR MAN M5 FWD
LD TR0
AND 10.09  ; IR HMI PB RVS MOTOR 5
OUT 14.09  ; IR MAN M5 RVS
LD TR0
AND 10.10  ; IR HMI PB STP1 UP
OUT 14.10  ; IR MAN STP1 UP
LD TR0
AND 10.11  ; IR HMI PB STP1 DN
OUT 14.11  ; IR MAN STP1 DN
LD TR0
AND 10.12  ; IR HMI PB STP2 UP
OUT 14.12  ; IR MAN STP2 UP
LD TR0
AND 10.13  ; IR HMI PB STP2 DN
OUT 14.13  ; IR MAN STP2 DN
LD TR0
AND 10.14  ; IR HMI PB STP3 UP
OUT 14.14  ; IR MAN STP3 UP
LD TR0
AND 10.15  ; IR HMI PB STP3 DN
AND 1.15  ; LS STRAIGHT
OUT 14.15  ; IR MAN STP3 DN
LD TR0
AND 18.02  ; IR HMI PB STP ROT UP
OUT 18.04  ; IR MAN STP ROT UP
LD TR0
AND 18.03  ; IR HMI STP ROT DN
OUT 18.05  ; IR MAN STP ROT DN
LD TR0
AND 19.07  ; IR HMI PB M ROLLER RVS
OUT 19.04  ; IR MAN M ROLLER RVS
LD TR0
AND 19.06  ; IR HMI PB M ROLLER FWD
OUT 19.05  ; IR MAN M ROLLER FWD
LD TR0
LD 10.04  ; IR HMI PB STRAIGHT
OR 19.14  ; SET HOMEPOST ALL
ANDLD
AND 1.13  ; RS DN STP ROTARY
ANDNOT 19.08  ; SET LS STRAIGHT
ANDNOT 1.15  ; LS STRAIGHT
OUT 14.04  ; IR MAN STRAIGHT ROT
LD TR0
AND 10.05  ; IR HMI PB TURN
AND 1.13  ; RS DN STP ROTARY
ANDNOT 19.09  ; SET LS TURN
ANDNOT 1.14  ; LS TURN
OUT 14.05  ; IR MAN TURN ROT

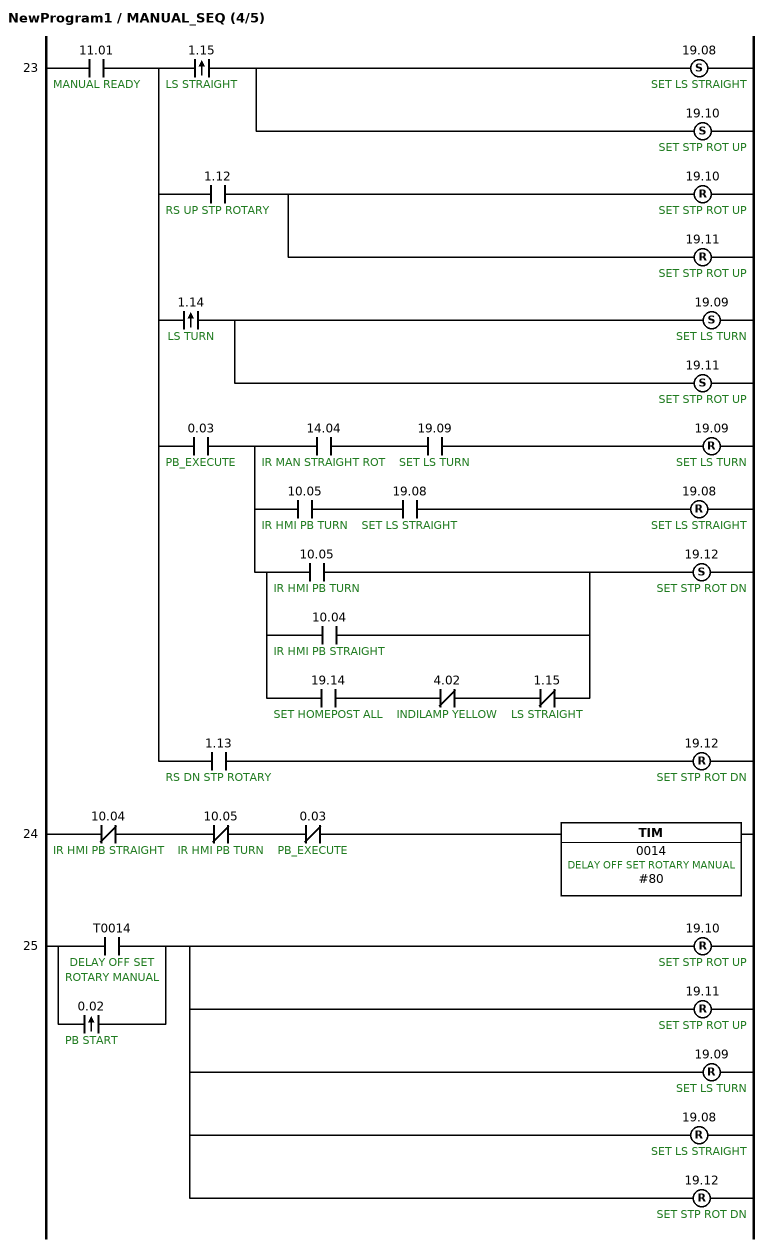
; rung 23
LD 11.01  ; MANUAL READY
OUT TR0
@AND 1.15  ; LS STRAIGHT
SET 19.08  ; SET LS STRAIGHT
SET 19.10  ; SET STP ROT UP
LD TR0
AND 1.12  ; RS UP STP ROTARY
RSET 19.10  ; SET STP ROT UP
RSET 19.11  ; SET STP ROT UP
LD TR0
@AND 1.14  ; LS TURN
SET 19.09  ; SET LS TURN
SET 19.11  ; SET STP ROT UP
LD TR0
AND 0.03  ; PB_EXECUTE
OUT TR1
AND 14.04  ; IR MAN STRAIGHT ROT
AND 19.09  ; SET LS TURN
RSET 19.09  ; SET LS TURN
LD TR1
AND 10.05  ; IR HMI PB TURN
AND 19.08  ; SET LS STRAIGHT
RSET 19.08  ; SET LS STRAIGHT
LD TR1
LD 10.05  ; IR HMI PB TURN
OR 10.04  ; IR HMI PB STRAIGHT
LD 19.14  ; SET HOMEPOST ALL
ANDNOT 4.02  ; INDILAMP YELLOW
ANDNOT 1.15  ; LS STRAIGHT
ORLD
ANDLD
SET 19.12  ; SET STP ROT DN
LD TR0
AND 1.13  ; RS DN STP ROTARY
RSET 19.12  ; SET STP ROT DN
; rung 24
LDNOT 10.04  ; IR HMI PB STRAIGHT
ANDNOT 10.05  ; IR HMI PB TURN
ANDNOT 0.03  ; PB_EXECUTE
TIM 0014 #80  ; DELAY OFF SET ROTARY MANUAL
; rung 25
LD T0014  ; DELAY OFF SET ROTARY MANUAL
@OR 0.02  ; PB START
RSET 19.10  ; SET STP ROT UP
RSET 19.11  ; SET STP ROT UP
RSET 19.09  ; SET LS TURN
RSET 19.08  ; SET LS STRAIGHT
RSET 19.12  ; SET STP ROT DN

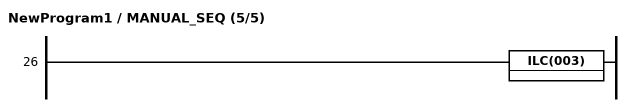
; rung 26
ILC(003)

### Section AUTO_SEQUENCE

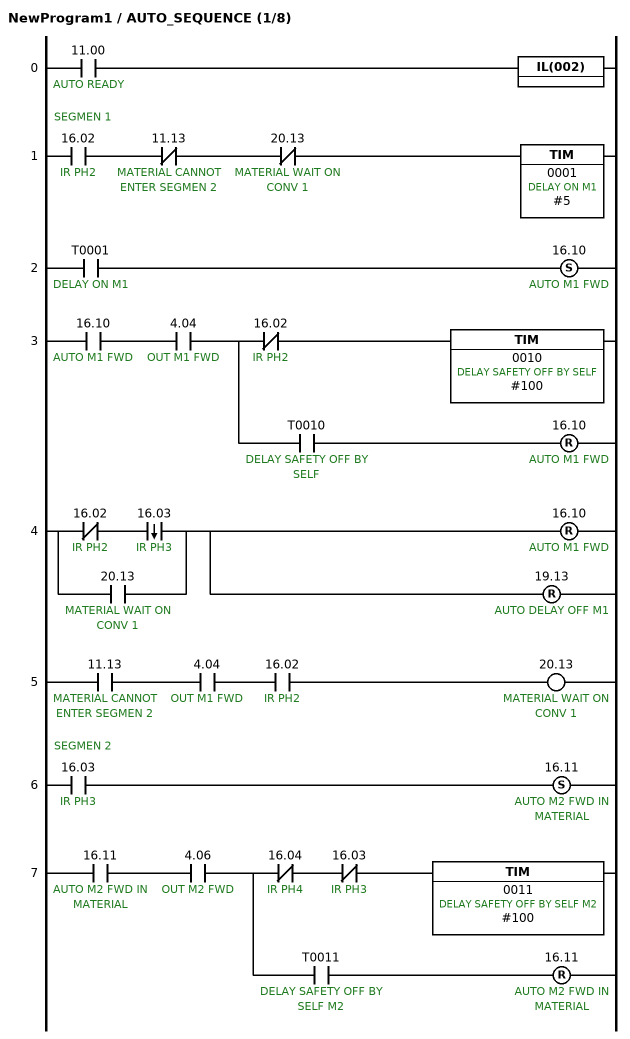
; rung 0
LD 11.00  ; AUTO READY
IL(002)
; rung 1: SEGMEN 1
LD 16.02  ; IR PH2
ANDNOT 11.13  ; MATERIAL CANNOT ENTER SEGMEN 2
ANDNOT 20.13  ; MATERIAL WAIT ON CONV 1
TIM 0001 #5  ; DELAY ON M1
; rung 2
LD T0001  ; DELAY ON M1
SET 16.10  ; AUTO M1 FWD
; rung 3
LD 16.10  ; AUTO M1 FWD
AND 4.04  ; OUT M1 FWD
OUT TR0
ANDNOT 16.02  ; IR PH2
TIM 0010 #100  ; DELAY SAFETY OFF BY SELF
LD TR0
AND T0010  ; DELAY SAFETY OFF BY SELF
RSET 16.10  ; AUTO M1 FWD
; rung 4
LDNOT 16.02  ; IR PH2
%AND 16.03  ; IR PH3
OR 20.13  ; MATERIAL WAIT ON CONV 1
RSET 16.10  ; AUTO M1 FWD
RSET 19.13  ; AUTO DELAY OFF M1
; rung 5
LD 11.13  ; MATERIAL CANNOT ENTER SEGMEN 2
AND 4.04  ; OUT M1 FWD
AND 16.02  ; IR PH2
OUT 20.13  ; MATERIAL WAIT ON CONV 1
; rung 6: SEGMEN 2
LD 16.03  ; IR PH3
SET 16.11  ; AUTO M2 FWD IN MATERIAL
; rung 7
LD 16.11  ; AUTO M2 FWD IN MATERIAL
AND 4.06  ; OUT M2 FWD
OUT TR0
ANDNOT 16.04  ; IR PH4
ANDNOT 16.03  ; IR PH3
TIM 0011 #100  ; DELAY SAFETY OFF BY SELF M2
LD TR0
AND T0011  ; DELAY SAFETY OFF BY SELF M2
RSET 16.11  ; AUTO M2 FWD IN MATERIAL

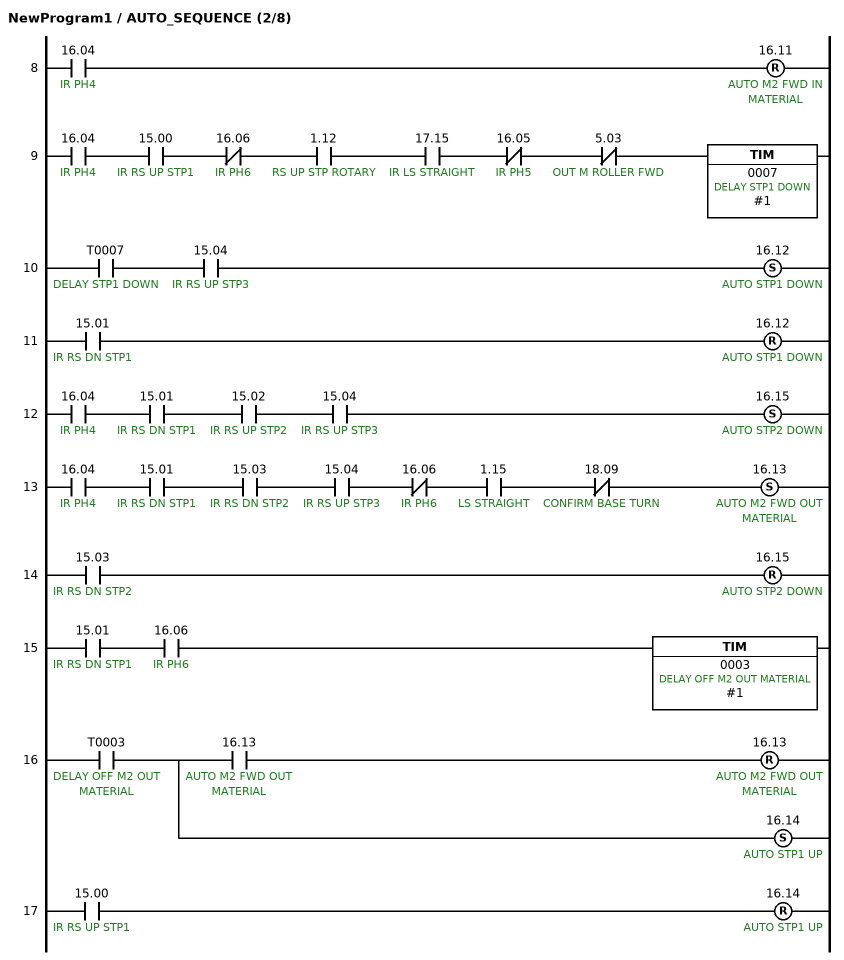
; rung 8
LD 16.04  ; IR PH4
RSET 16.11  ; AUTO M2 FWD IN MATERIAL
; rung 9
LD 16.04  ; IR PH4
AND 15.00  ; IR RS UP STP1
ANDNOT 16.06  ; IR PH6
AND 1.12  ; RS UP STP ROTARY
AND 17.15  ; IR LS STRAIGHT
ANDNOT 16.05  ; IR PH5
ANDNOT 5.03  ; OUT M ROLLER FWD
TIM 0007 #1  ; DELAY STP1 DOWN
; rung 10
LD T0007  ; DELAY STP1 DOWN
AND 15.04  ; IR RS UP STP3
SET 16.12  ; AUTO STP1 DOWN
; rung 11
LD 15.01  ; IR RS DN STP1
RSET 16.12  ; AUTO STP1 DOWN
; rung 12
LD 16.04  ; IR PH4
AND 15.01  ; IR RS DN STP1
AND 15.02  ; IR RS UP STP2
AND 15.04  ; IR RS UP STP3
SET 16.15  ; AUTO STP2 DOWN
; rung 13
LD 16.04  ; IR PH4
AND 15.01  ; IR RS DN STP1
AND 15.03  ; IR RS DN STP2
AND 15.04  ; IR RS UP STP3
ANDNOT 16.06  ; IR PH6
AND 1.15  ; LS STRAIGHT
ANDNOT 18.09  ; CONFIRM BASE TURN
SET 16.13  ; AUTO M2 FWD OUT MATERIAL
; rung 14
LD 15.03  ; IR RS DN STP2
RSET 16.15  ; AUTO STP2 DOWN
; rung 15
LD 15.01  ; IR RS DN STP1
AND 16.06  ; IR PH6
TIM 0003 #1  ; DELAY OFF M2 OUT MATERIAL
; rung 16
LD T0003  ; DELAY OFF M2 OUT MATERIAL
OUT TR0
AND 16.13  ; AUTO M2 FWD OUT MATERIAL
RSET 16.13  ; AUTO M2 FWD OUT MATERIAL
LD TR0
SET 16.14  ; AUTO STP1 UP
; rung 17
LD 15.00  ; IR RS UP STP1
RSET 16.14  ; AUTO STP1 UP

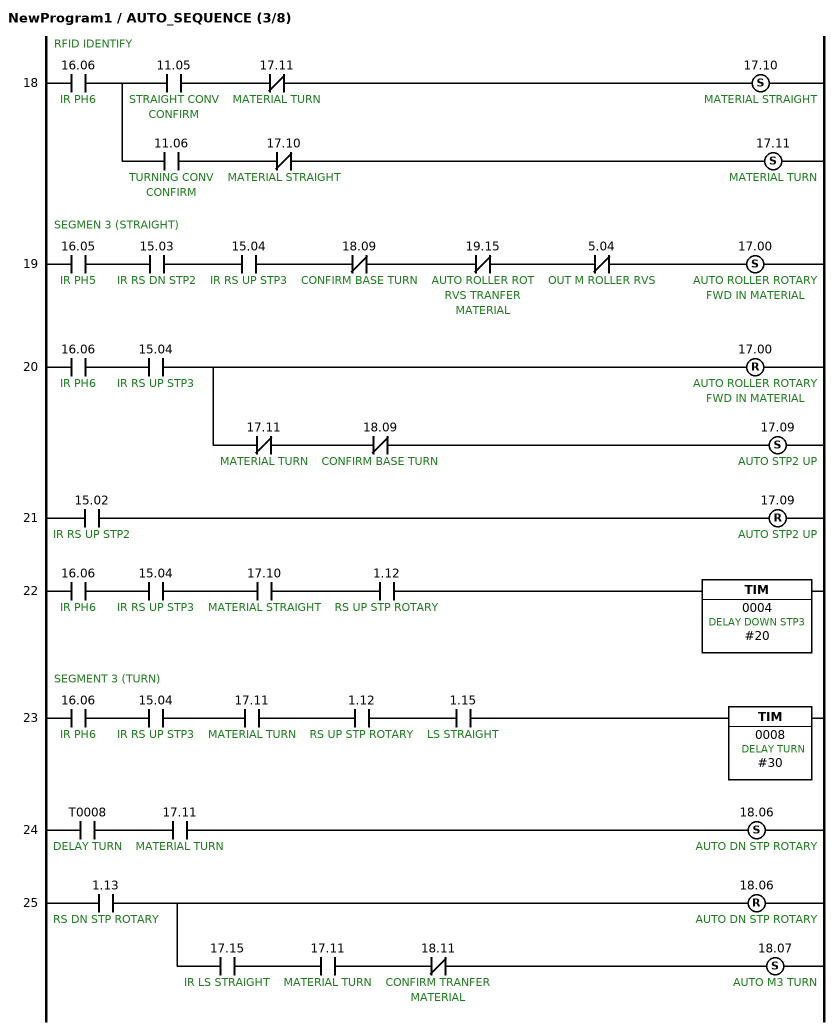
; rung 18: RFID IDENTIFY
LD 16.06  ; IR PH6
OUT TR0
AND 11.05  ; STRAIGHT CONV CONFIRM
ANDNOT 17.11  ; MATERIAL TURN
SET 17.10  ; MATERIAL STRAIGHT
LD TR0
AND 11.06  ; TURNING CONV CONFIRM
ANDNOT 17.10  ; MATERIAL STRAIGHT
SET 17.11  ; MATERIAL TURN
; rung 19: SEGMEN 3 (STRAIGHT)
LD 16.05  ; IR PH5
AND 15.03  ; IR RS DN STP2
AND 15.04  ; IR RS UP STP3
ANDNOT 18.09  ; CONFIRM BASE TURN
ANDNOT 19.15  ; AUTO ROLLER ROT RVS TRANFER MATERIAL
ANDNOT 5.04  ; OUT M ROLLER RVS
SET 17.00  ; AUTO ROLLER ROTARY FWD IN MATERIAL
; rung 20
LD 16.06  ; IR PH6
AND 15.04  ; IR RS UP STP3
RSET 17.00  ; AUTO ROLLER ROTARY FWD IN MATERIAL
ANDNOT 17.11  ; MATERIAL TURN
ANDNOT 18.09  ; CONFIRM BASE TURN
SET 17.09  ; AUTO STP2 UP
; rung 21
LD 15.02  ; IR RS UP STP2
RSET 17.09  ; AUTO STP2 UP
; rung 22
LD 16.06  ; IR PH6
AND 15.04  ; IR RS UP STP3
AND 17.10  ; MATERIAL STRAIGHT
AND 1.12  ; RS UP STP ROTARY
TIM 0004 #20  ; DELAY DOWN STP3
; rung 23: SEGMENT 3 (TURN)
LD 16.06  ; IR PH6
AND 15.04  ; IR RS UP STP3
AND 17.11  ; MATERIAL TURN
AND 1.12  ; RS UP STP ROTARY
AND 1.15  ; LS STRAIGHT
TIM 0008 #30  ; DELAY TURN
; rung 24
LD T0008  ; DELAY TURN
AND 17.11  ; MATERIAL TURN
SET 18.06  ; AUTO DN STP ROTARY
; rung 25
LD 1.13  ; RS DN STP ROTARY
RSET 18.06  ; AUTO DN STP ROTARY
AND 17.15  ; IR LS STRAIGHT
AND 17.11  ; MATERIAL TURN
ANDNOT 18.11  ; CONFIRM TRANFER MATERIAL
SET 18.07  ; AUTO M3 TURN

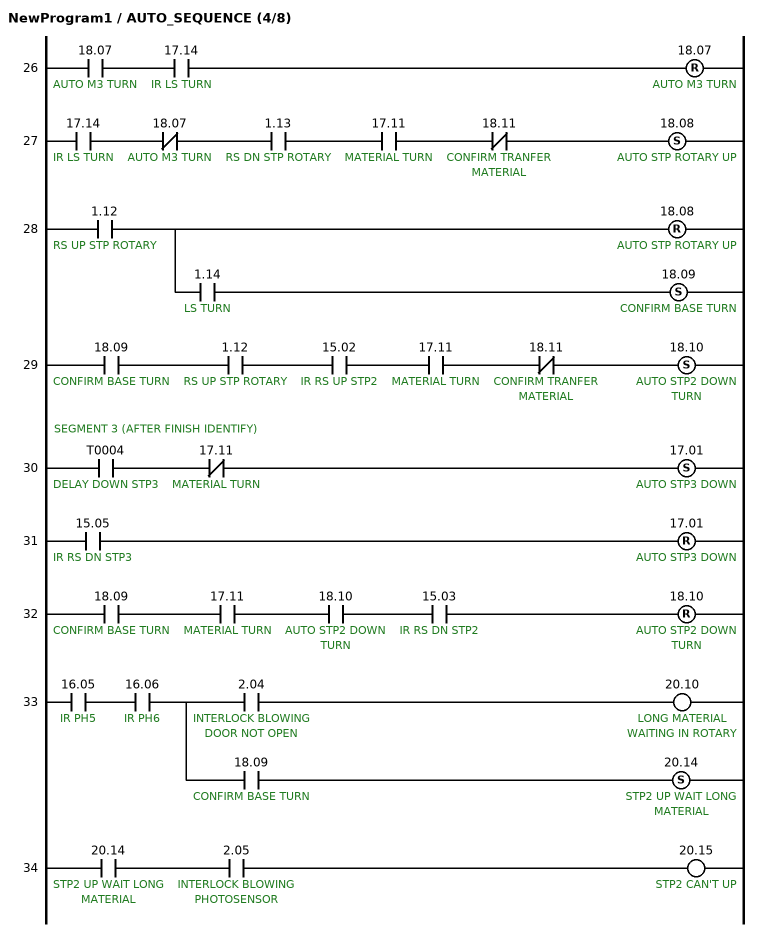
; rung 26
LD 18.07  ; AUTO M3 TURN
AND 17.14  ; IR LS TURN
RSET 18.07  ; AUTO M3 TURN
; rung 27
LD 17.14  ; IR LS TURN
ANDNOT 18.07  ; AUTO M3 TURN
AND 1.13  ; RS DN STP ROTARY
AND 17.11  ; MATERIAL TURN
ANDNOT 18.11  ; CONFIRM TRANFER MATERIAL
SET 18.08  ; AUTO STP ROTARY UP
; rung 28
LD 1.12  ; RS UP STP ROTARY
RSET 18.08  ; AUTO STP ROTARY UP
AND 1.14  ; LS TURN
SET 18.09  ; CONFIRM BASE TURN
; rung 29
LD 18.09  ; CONFIRM BASE TURN
AND 1.12  ; RS UP STP ROTARY
AND 15.02  ; IR RS UP STP2
AND 17.11  ; MATERIAL TURN
ANDNOT 18.11  ; CONFIRM TRANFER MATERIAL
SET 18.10  ; AUTO STP2 DOWN TURN
; rung 30: SEGMENT 3 (AFTER FINISH IDENTIFY)
LD T0004  ; DELAY DOWN STP3
ANDNOT 17.11  ; MATERIAL TURN
SET 17.01  ; AUTO STP3 DOWN
; rung 31
LD 15.05  ; IR RS DN STP3
RSET 17.01  ; AUTO STP3 DOWN
; rung 32
LD 18.09  ; CONFIRM BASE TURN
AND 17.11  ; MATERIAL TURN
AND 18.10  ; AUTO STP2 DOWN TURN
AND 15.03  ; IR RS DN STP2
RSET 18.10  ; AUTO STP2 DOWN TURN
; rung 33
LD 16.05  ; IR PH5
AND 16.06  ; IR PH6
OUT TR0
AND 2.04  ; INTERLOCK BLOWING DOOR NOT OPEN
OUT 20.10  ; LONG MATERIAL WAITING IN ROTARY
LD TR0
AND 18.09  ; CONFIRM BASE TURN
SET 20.14  ; STP2 UP WAIT LONG MATERIAL
; rung 34
LD 20.14  ; STP2 UP WAIT LONG MATERIAL
AND 2.05  ; INTERLOCK BLOWING PHOTOSENSOR
OUT 20.15  ; STP2 CAN'T UP

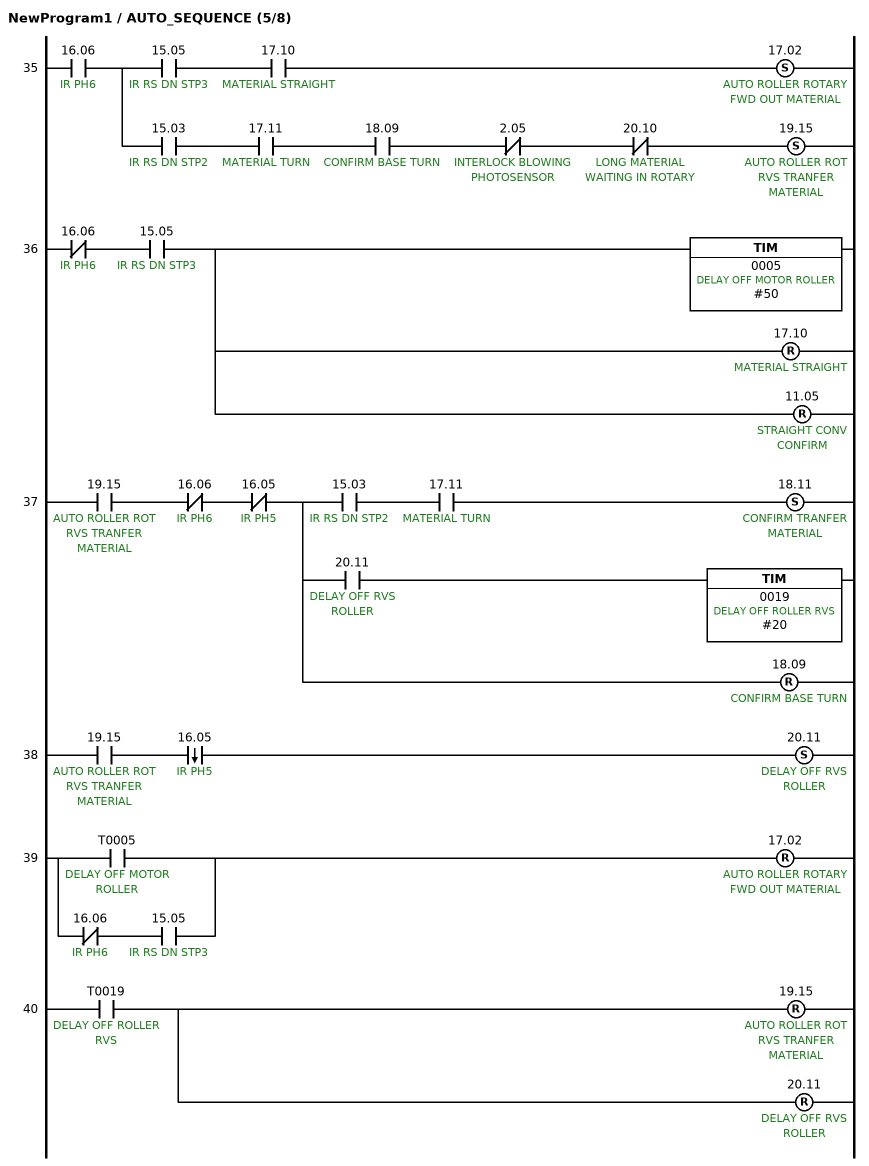
; rung 35
LD 16.06  ; IR PH6
OUT TR0
AND 15.05  ; IR RS DN STP3
AND 17.10  ; MATERIAL STRAIGHT
SET 17.02  ; AUTO ROLLER ROTARY FWD OUT MATERIAL
LD TR0
AND 15.03  ; IR RS DN STP2
AND 17.11  ; MATERIAL TURN
AND 18.09  ; CONFIRM BASE TURN
ANDNOT 2.05  ; INTERLOCK BLOWING PHOTOSENSOR
ANDNOT 20.10  ; LONG MATERIAL WAITING IN ROTARY
SET 19.15  ; AUTO ROLLER ROT RVS TRANFER MATERIAL
; rung 36
LDNOT 16.06  ; IR PH6
AND 15.05  ; IR RS DN STP3
TIM 0005 #50  ; DELAY OFF MOTOR ROLLER
RSET 17.10  ; MATERIAL STRAIGHT
RSET 11.05  ; STRAIGHT CONV CONFIRM
; rung 37
LD 19.15  ; AUTO ROLLER ROT RVS TRANFER MATERIAL
ANDNOT 16.06  ; IR PH6
ANDNOT 16.05  ; IR PH5
OUT TR0
AND 15.03  ; IR RS DN STP2
AND 17.11  ; MATERIAL TURN
SET 18.11  ; CONFIRM TRANFER MATERIAL
LD TR0
AND 20.11  ; DELAY OFF RVS ROLLER
TIM 0019 #20  ; DELAY OFF ROLLER RVS
LD TR0
RSET 18.09  ; CONFIRM BASE TURN
; rung 38
LD 19.15  ; AUTO ROLLER ROT RVS TRANFER MATERIAL
%AND 16.05  ; IR PH5
SET 20.11  ; DELAY OFF RVS ROLLER
; rung 39
LD T0005  ; DELAY OFF MOTOR ROLLER
LDNOT 16.06  ; IR PH6
AND 15.05  ; IR RS DN STP3
ORLD
RSET 17.02  ; AUTO ROLLER ROTARY FWD OUT MATERIAL
; rung 40
LD T0019  ; DELAY OFF ROLLER RVS
RSET 19.15  ; AUTO ROLLER ROT RVS TRANFER MATERIAL
RSET 20.11  ; DELAY OFF RVS ROLLER

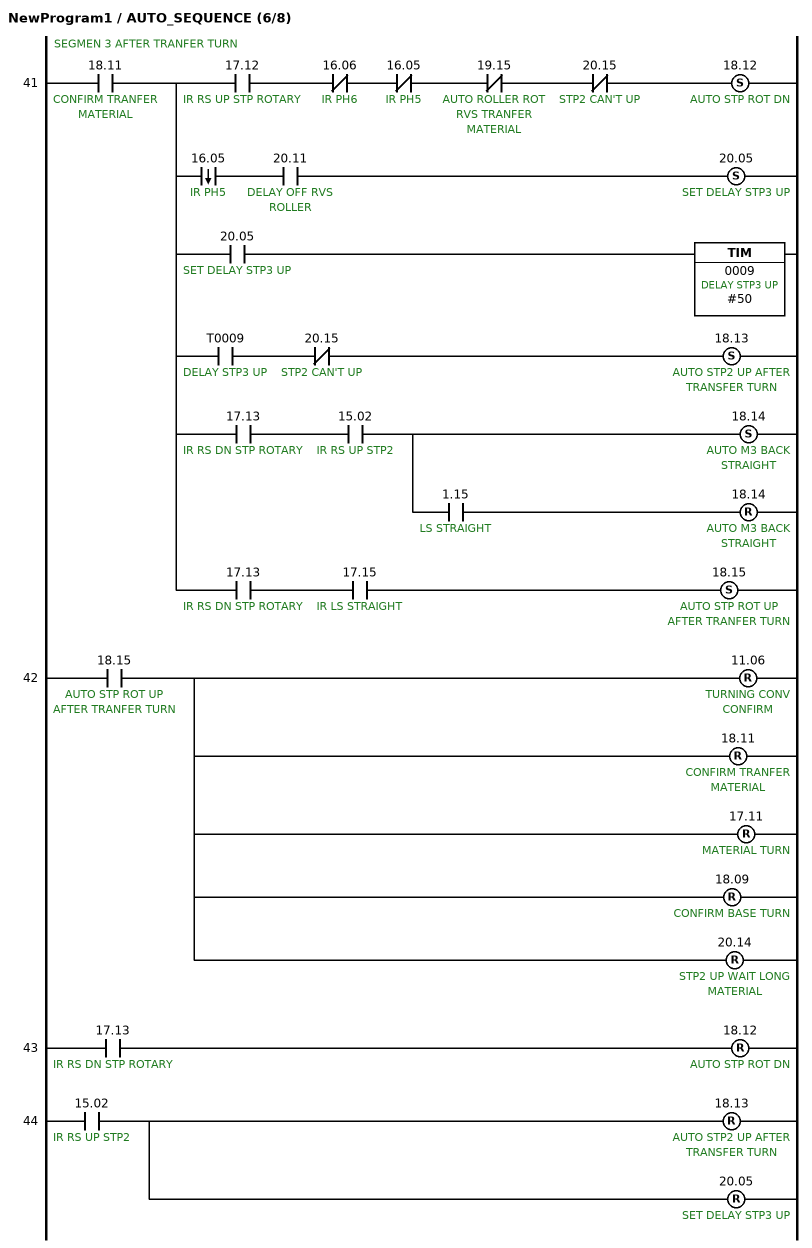
; rung 41: SEGMEN 3 AFTER TRANFER TURN
LD 18.11  ; CONFIRM TRANFER MATERIAL
OUT TR0
AND 17.12  ; IR RS UP STP ROTARY
ANDNOT 16.06  ; IR PH6
ANDNOT 16.05  ; IR PH5
ANDNOT 19.15  ; AUTO ROLLER ROT RVS TRANFER MATERIAL
ANDNOT 20.15  ; STP2 CAN'T UP
SET 18.12  ; AUTO STP ROT DN
LD TR0
%AND 16.05  ; IR PH5
AND 20.11  ; DELAY OFF RVS ROLLER
SET 20.05  ; SET DELAY STP3 UP
LD TR0
AND 20.05  ; SET DELAY STP3 UP
TIM 0009 #50  ; DELAY STP3 UP
LD TR0
AND T0009  ; DELAY STP3 UP
ANDNOT 20.15  ; STP2 CAN'T UP
SET 18.13  ; AUTO STP2 UP AFTER TRANSFER TURN
LD TR0
AND 17.13  ; IR RS DN STP ROTARY
AND 15.02  ; IR RS UP STP2
SET 18.14  ; AUTO M3 BACK STRAIGHT
AND 1.15  ; LS STRAIGHT
RSET 18.14  ; AUTO M3 BACK STRAIGHT
LD TR0
AND 17.13  ; IR RS DN STP ROTARY
AND 17.15  ; IR LS STRAIGHT
SET 18.15  ; AUTO STP ROT UP AFTER TRANFER TURN
; rung 42
LD 18.15  ; AUTO STP ROT UP AFTER TRANFER TURN
RSET 11.06  ; TURNING CONV CONFIRM
RSET 18.11  ; CONFIRM TRANFER MATERIAL
RSET 17.11  ; MATERIAL TURN
RSET 18.09  ; CONFIRM BASE TURN
RSET 20.14  ; STP2 UP WAIT LONG MATERIAL
; rung 43
LD 17.13  ; IR RS DN STP ROTARY
RSET 18.12  ; AUTO STP ROT DN
; rung 44
LD 15.02  ; IR RS UP STP2
RSET 18.13  ; AUTO STP2 UP AFTER TRANSFER TURN
RSET 20.05  ; SET DELAY STP3 UP

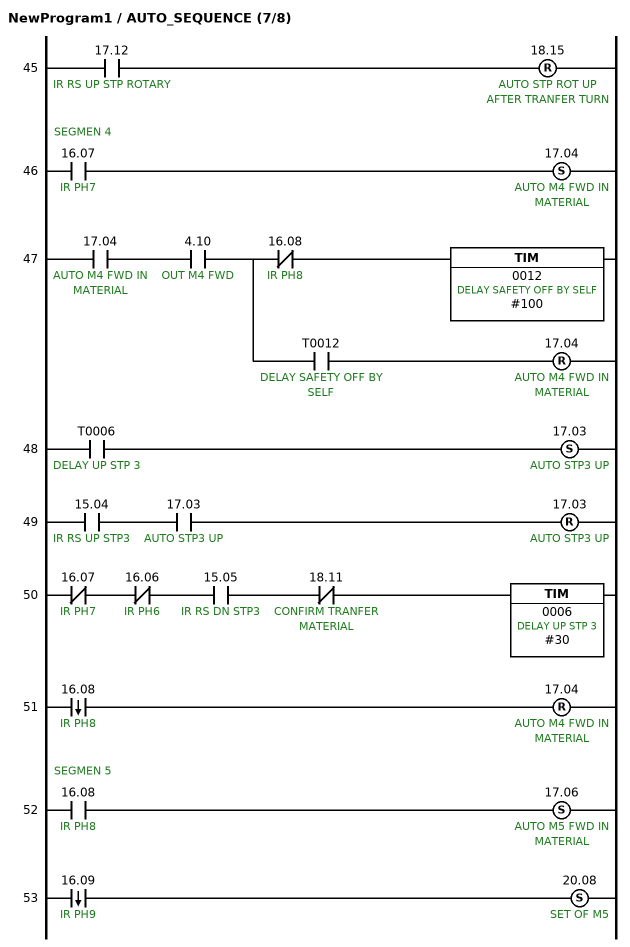
; rung 45
LD 17.12  ; IR RS UP STP ROTARY
RSET 18.15  ; AUTO STP ROT UP AFTER TRANFER TURN
; rung 46: SEGMEN 4
LD 16.07  ; IR PH7
SET 17.04  ; AUTO M4 FWD IN MATERIAL
; rung 47
LD 17.04  ; AUTO M4 FWD IN MATERIAL
AND 4.10  ; OUT M4 FWD
OUT TR0
ANDNOT 16.08  ; IR PH8
TIM 0012 #100  ; DELAY SAFETY OFF BY SELF
LD TR0
AND T0012  ; DELAY SAFETY OFF BY SELF
RSET 17.04  ; AUTO M4 FWD IN MATERIAL
; rung 48
LD T0006  ; DELAY UP STP 3
SET 17.03  ; AUTO STP3 UP
; rung 49
LD 15.04  ; IR RS UP STP3
AND 17.03  ; AUTO STP3 UP
RSET 17.03  ; AUTO STP3 UP
; rung 50
LDNOT 16.07  ; IR PH7
ANDNOT 16.06  ; IR PH6
AND 15.05  ; IR RS DN STP3
ANDNOT 18.11  ; CONFIRM TRANFER MATERIAL
TIM 0006 #30  ; DELAY UP STP 3
; rung 51
%LD 16.08  ; IR PH8
RSET 17.04  ; AUTO M4 FWD IN MATERIAL
; rung 52: SEGMEN 5
LD 16.08  ; IR PH8
SET 17.06  ; AUTO M5 FWD IN MATERIAL
; rung 53
%LD 16.09  ; IR PH9
SET 20.08  ; SET OF M5

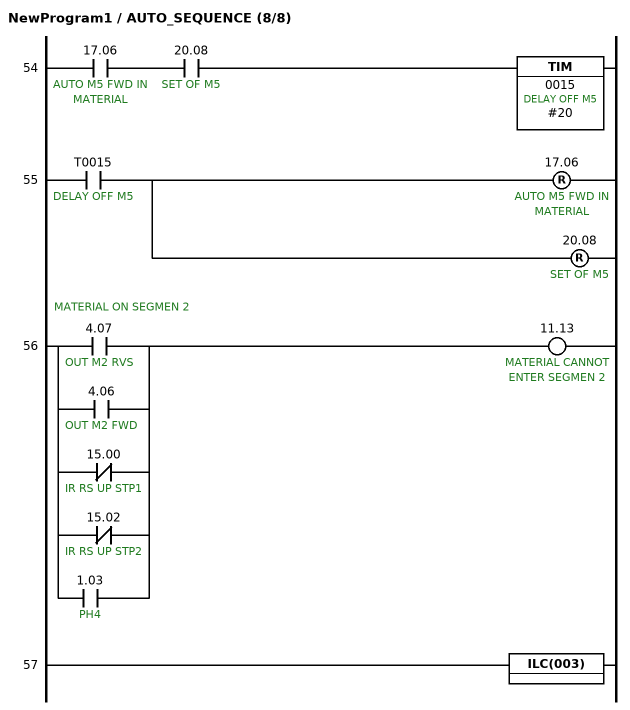
; rung 54
LD 17.06  ; AUTO M5 FWD IN MATERIAL
AND 20.08  ; SET OF M5
TIM 0015 #20  ; DELAY OFF M5
; rung 55
LD T0015  ; DELAY OFF M5
RSET 17.06  ; AUTO M5 FWD IN MATERIAL
RSET 20.08  ; SET OF M5
; rung 56: MATERIAL ON SEGMEN 2
LD 4.07  ; OUT M2 RVS
OR 4.06  ; OUT M2 FWD
ORNOT 15.00  ; IR RS UP STP1
ORNOT 15.02  ; IR RS UP STP2
OR 1.03  ; PH4
OUT 11.13  ; MATERIAL CANNOT ENTER SEGMEN 2
; rung 57
ILC(003)

### Section OUTPUT_REAL

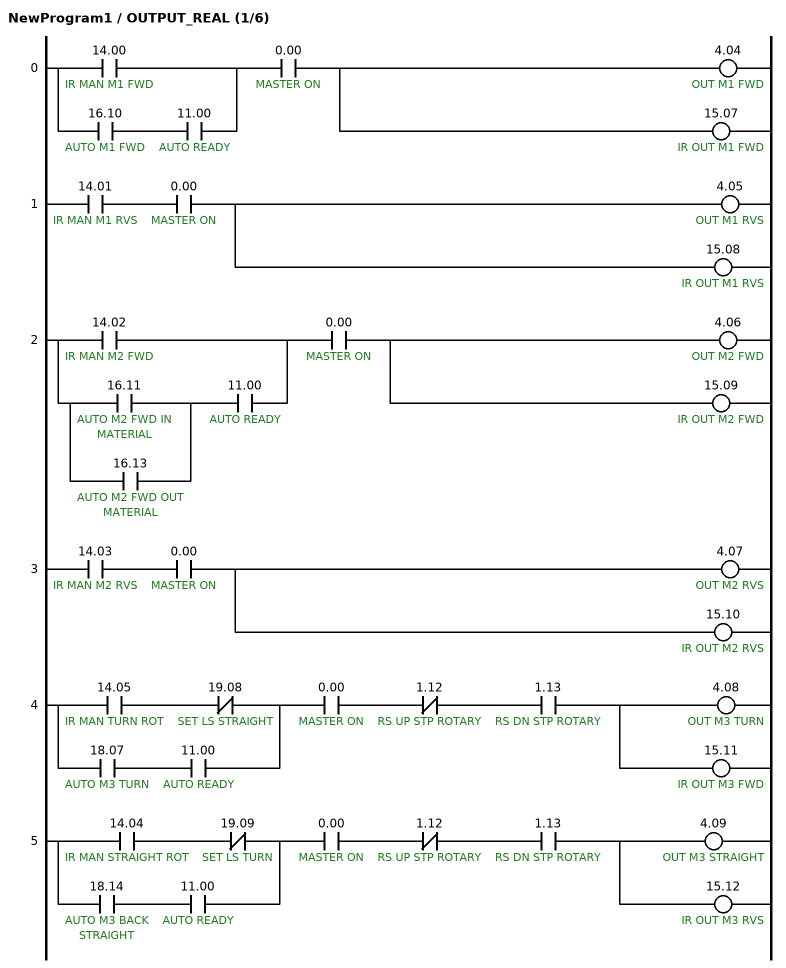
; rung 0
LD 14.00  ; IR MAN M1 FWD
LD 16.10  ; AUTO M1 FWD
AND 11.00  ; AUTO READY
ORLD
AND 0.00  ; MASTER ON
OUT 4.04  ; OUT M1 FWD
OUT 15.07  ; IR OUT M1 FWD
; rung 1
LD 14.01  ; IR MAN M1 RVS
AND 0.00  ; MASTER ON
OUT 4.05  ; OUT M1 RVS
OUT 15.08  ; IR OUT M1 RVS
; rung 2
LD 14.02  ; IR MAN M2 FWD
LD 16.11  ; AUTO M2 FWD IN MATERIAL
OR 16.13  ; AUTO M2 FWD OUT MATERIAL
AND 11.00  ; AUTO READY
ORLD
AND 0.00  ; MASTER ON
OUT 4.06  ; OUT M2 FWD
OUT 15.09  ; IR OUT M2 FWD
; rung 3
LD 14.03  ; IR MAN M2 RVS
AND 0.00  ; MASTER ON
OUT 4.07  ; OUT M2 RVS
OUT 15.10  ; IR OUT M2 RVS
; rung 4
LD 14.05  ; IR MAN TURN ROT
ANDNOT 19.08  ; SET LS STRAIGHT
LD 18.07  ; AUTO M3 TURN
AND 11.00  ; AUTO READY
ORLD
AND 0.00  ; MASTER ON
ANDNOT 1.12  ; RS UP STP ROTARY
AND 1.13  ; RS DN STP ROTARY
OUT 4.08  ; OUT M3 TURN
OUT 15.11  ; IR OUT M3 FWD
; rung 5
LD 14.04  ; IR MAN STRAIGHT ROT
ANDNOT 19.09  ; SET LS TURN
LD 18.14  ; AUTO M3 BACK STRAIGHT
AND 11.00  ; AUTO READY
ORLD
AND 0.00  ; MASTER ON
ANDNOT 1.12  ; RS UP STP ROTARY
AND 1.13  ; RS DN STP ROTARY
OUT 4.09  ; OUT M3 STRAIGHT
OUT 15.12  ; IR OUT M3 RVS

